	1: (* GET CLIMATIC *)
		Cmd_RLen:=20;
		FOR i:=0 TO 4 DO
			j:=DINT_TO_INT(CAL01_Clima.Points[i].X);
			TxLen:=TxLen+RAWTOHEX(ADR(j),2,ADR(TxData[TxLen]));
			j:=DINT_TO_INT(CAL01_Clima.Points[i].Y);
			TxLen:=TxLen+RAWTOHEX(ADR(j),2,ADR(TxData[TxLen]));
		END_FOR

	2: (* SET CLIMATIC *)
		IF Cmd_CLen<>20 THEN
			Cmd_R:=4;
		ELSE
			FOR i:=0 TO 4 DO
				Cmd_Buf_INT:=ADR(Cmd_Buf[8+4*i]); j:=Cmd_Buf_INT^;
				CAL01_Clima.Points[i].X:=INT_TO_DINT(j);
				Cmd_Buf_INT:=ADR(Cmd_Buf[10+4*i]); j:=Cmd_Buf_INT^;
				CAL01_Clima.Points[i].Y:=INT_TO_DINT(j);
			END_FOR
		END_IF




ELSE
	Cmd_R:=3;
END_CASE
END_ACTION
ACTION Cmd_CIR:
IF Cmd_ObjIdx<1 OR Cmd_ObjIdx>6 THEN
	Cmd_R:=2;
	RETURN;
END_IF

(* Process command *)
CASE Cmd_C OF

	1:	(* Force CIR On *)
		CASE Cmd_ObjIdx OF

		(*	1:	CIR01.CIR_RUN_REQ := TRUE; *)
			2:	CIR02.CIR_RUN_REQ := TRUE;
			3:	CIR03.CIR_RUN_REQ := TRUE;
			4:	CIR04.CIR_RUN_REQ := TRUE;
			5:	CIR05.CIR_RUN_REQ := TRUE;
			6:	CIR06.CIR_RUN_REQ := TRUE;

		END_CASE

	2:	(* Force CIR Off *)
		CASE Cmd_ObjIdx OF

		(*	1:	CIR01.CIR_STOP_REQ := TRUE; *)
			2:	CIR02.CIR_STOP_REQ := TRUE;
			3:	CIR03.CIR_STOP_REQ := TRUE;
			4:	CIR04.CIR_STOP_REQ := TRUE;
			5:	CIR05.CIR_STOP_REQ := TRUE;
			6:	CIR06.CIR_STOP_REQ := TRUE;

		END_CASE

	3:	(* Release force *)
		CASE Cmd_ObjIdx OF

		(*	1:	CIR01.CIR_RUN_REQ	:= FALSE;
				CIR01.CIR_STOP_REQ 	:= FALSE; *)
			2:	CIR02.CIR_RUN_REQ	:= FALSE;
				CIR02.CIR_STOP_REQ 	:= FALSE;
			3:	CIR03.CIR_RUN_REQ	:= FALSE;
				CIR03.CIR_STOP_REQ 	:= FALSE;
			4:	CIR04.CIR_RUN_REQ	:= FALSE;
				CIR04.CIR_STOP_REQ 	:= FALSE;
			5:	CIR05.CIR_RUN_REQ	:= FALSE;
				CIR05.CIR_STOP_REQ 	:= FALSE;
			6:	CIR06.CIR_RUN_REQ	:= FALSE;
				CIR06.CIR_STOP_REQ 	:= FALSE;

		END_CASE


	4: (* SET Tempi delay On Off Circolatori  *)
		CASE Cmd_ObjIdx OF
		(*	1:	Cmd_Buf_U16:=ADR(Cmd_Buf[8]);
				CIR01.OnDelay := DWORD_TO_TIME((Cmd_Buf_U16^)*60*1000); 			(* Delay ON*)
				Cmd_Buf_U16:=ADR(Cmd_Buf[10]);
				CIR01.OffDelay := DWORD_TO_TIME((Cmd_Buf_U16^)*60*1000);			(* Delay OFF *) *)

			2:	Cmd_Buf_U16:=ADR(Cmd_Buf[8]);
				CIR02.OnDelay := DWORD_TO_TIME((Cmd_Buf_U16^)*60*1000);			(* Delay ON*)
				Cmd_Buf_U16:=ADR(Cmd_Buf[10]);
				CIR02.OffDelay := DWORD_TO_TIME((Cmd_Buf_U16^)*60*1000);			(* Delay OFF *)

			3:	Cmd_Buf_U16:=ADR(Cmd_Buf[8]);
				CIR03.OnDelay := DWORD_TO_TIME((Cmd_Buf_U16^)*60*1000); 			(* Delay ON*)
				Cmd_Buf_U16:=ADR(Cmd_Buf[10]);
				CIR03.OffDelay := DWORD_TO_TIME((Cmd_Buf_U16^)*60*1000);			(* Delay OFF *)

			4:	Cmd_Buf_U16:=ADR(Cmd_Buf[8]);
				CIR04.OnDelay := DWORD_TO_TIME((Cmd_Buf_U16^)*60*1000);			(* Delay ON*)
				Cmd_Buf_U16:=ADR(Cmd_Buf[10]);
				CIR04.OffDelay := DWORD_TO_TIME((Cmd_Buf_U16^)*60*1000);			(* Delay OFF *)

			5:	Cmd_Buf_U16:=ADR(Cmd_Buf[8]);
				CIR05.OnDelay := DWORD_TO_TIME((Cmd_Buf_U16^)*60*1000); 			(* Delay ON*)
				Cmd_Buf_U16:=ADR(Cmd_Buf[10]);
				CIR05.OffDelay := DWORD_TO_TIME((Cmd_Buf_U16^)*60*1000);			(* Delay OFF *)

			6:	Cmd_Buf_U16:=ADR(Cmd_Buf[8]);
				CIR06.OnDelay := DWORD_TO_TIME((Cmd_Buf_U16^)*60*1000);			(* Delay ON*)
				Cmd_Buf_U16:=ADR(Cmd_Buf[10]);
				CIR06.OffDelay := DWORD_TO_TIME((Cmd_Buf_U16^)*60*1000);			(* Delay OFF *)

		END_CASE


	5: (* GET Tempi delay On Off Circolatori *)
		Cmd_RLen:=4;
			CASE Cmd_ObjIdx OF


		(*	1:	j:=DWORD_TO_WORD(TIME_TO_DWORD((CIR01.OnDelay)/60/1000));
				TxLen:=TxLen+RAWTOHEX(ADR(j),2,ADR(TxData[TxLen]));
				j:=DWORD_TO_WORD(TIME_TO_DWORD((CIR01.OffDelay)/60/1000));
				TxLen:=TxLen+RAWTOHEX(ADR(j),2,ADR(TxData[TxLen]));   *)
			2: 	j:=DWORD_TO_WORD(TIME_TO_DWORD((CIR02.OnDelay)/60/1000));
				TxLen:=TxLen+RAWTOHEX(ADR(j),2,ADR(TxData[TxLen]));
				j:=DWORD_TO_WORD(TIME_TO_DWORD((CIR02.OffDelay)/60/1000));
				TxLen:=TxLen+RAWTOHEX(ADR(j),2,ADR(TxData[TxLen]));
			3:	j:=DWORD_TO_WORD(TIME_TO_DWORD((CIR03.OnDelay)/60/1000));
				TxLen:=TxLen+RAWTOHEX(ADR(j),2,ADR(TxData[TxLen]));
				j:=DWORD_TO_WORD(TIME_TO_DWORD((CIR03.OffDelay)/60/1000));
				TxLen:=TxLen+RAWTOHEX(ADR(j),2,ADR(TxData[TxLen]));
			4: 	j:=DWORD_TO_WORD(TIME_TO_DWORD((CIR04.OnDelay)/60/1000));
				TxLen:=TxLen+RAWTOHEX(ADR(j),2,ADR(TxData[TxLen]));
				j:=DWORD_TO_WORD(TIME_TO_DWORD((CIR04.OffDelay)/60/1000));
				TxLen:=TxLen+RAWTOHEX(ADR(j),2,ADR(TxData[TxLen]));
			5:	j:=DWORD_TO_WORD(TIME_TO_DWORD((CIR05.OnDelay)/60/1000));
				TxLen:=TxLen+RAWTOHEX(ADR(j),2,ADR(TxData[TxLen]));
				j:=DWORD_TO_WORD(TIME_TO_DWORD((CIR05.OffDelay)/60/1000));
				TxLen:=TxLen+RAWTOHEX(ADR(j),2,ADR(TxData[TxLen]));
			6: 	j:=DWORD_TO_WORD(TIME_TO_DWORD((CIR06.OnDelay)/60/1000));
				TxLen:=TxLen+RAWTOHEX(ADR(j),2,ADR(TxData[TxLen]));
				j:=DWORD_TO_WORD(TIME_TO_DWORD((CIR06.OffDelay)/60/1000));
				TxLen:=TxLen+RAWTOHEX(ADR(j),2,ADR(TxData[TxLen]));
		END_CASE










ELSE
	Cmd_R:=3;
END_CASE
END_ACTION
ACTION Cmd_CIRD:
IF Cmd_ObjIdx<1 OR Cmd_ObjIdx>2 THEN
	Cmd_R:=2;
	RETURN;
END_IF

(* Process command *)
CASE Cmd_C OF

	1:	(* Force CIR On *)
		CASE Cmd_ObjIdx OF

(*			1:	CIRD01.CIR_RUN_REQ := TRUE;
			2:	CIRD02.CIR_RUN_REQ := TRUE;
			3:	CIRD03.CIR_RUN_REQ := TRUE; *)

		END_CASE

	2:	(* Force CIR Off *)
		CASE Cmd_ObjIdx OF

(*			1:	CIRD01.CIR_STOP_REQ := TRUE;
			2:	CIRD02.CIR_STOP_REQ := TRUE;
			3:	CIRD03.CIR_STOP_REQ := TRUE; *)

		END_CASE

	3:	(* Release force *)
		CASE Cmd_ObjIdx OF

(*			1:	CIRD01.CIR_RUN_REQ	:= FALSE;
				CIRD01.CIR_STOP_REQ := FALSE;
			2:	CIRD02.CIR_RUN_REQ	:= FALSE;
				CIRD02.CIR_STOP_REQ := FALSE;
			3:	CIRD03.CIR_RUN_REQ 	:= FALSE;
				CIRD03.CIR_STOP_REQ := FALSE; *)

		END_CASE

ELSE
	Cmd_R:=3;
END_CASE
END_ACTION
ACTION Cmd_CRON:
(* Check index *)
IF Cmd_ObjIdx<1 OR Cmd_ObjIdx>6 THEN
	Cmd_R:=2;
	RETURN;
END_IF

(* Process command *)
CASE Cmd_C OF

	1: (* GET PROFILE *)
		IF Cmd_CLen<>3 THEN
			Cmd_R:=4;
		ELSE
			(* Load profile *)
			CronEd.CN_Sel:=WORD_TO_BYTE(Cmd_ObjIdx);
			Cmd_Buf_U16:=ADR(Cmd_Buf[8]);
			CronEd.CN_YSel:=Cmd_Buf_U16^;
			IF Cmd_Buf[10]<=10 THEN
				CronEd.PR_Sel:=Cmd_Buf[10];
				CronEd.PR_Load_Exe();
				(* Response data *)
				Cmd_RLen:=192;
				TxLen:=TxLen+RAWTOHEX(ADR(CronEd.PR.Setpoint),192,ADR(TxData[TxLen]));
			ELSE
				Cmd_R:=6;
			END_IF
		END_IF

	2: (* SET PROFILE *)
		IF Cmd_CLen<>(3+192) THEN
			Cmd_R:=4;
		ELSE
			(* Save profile *)
			CronEd.CN_Sel:=WORD_TO_BYTE(Cmd_ObjIdx);
			Cmd_Buf_U16:=ADR(Cmd_Buf[8]);
			CronEd.CN_YSel:=Cmd_Buf_U16^;
			IF Cmd_Buf[10]<=10 THEN
				CronEd.PR_Sel:=Cmd_Buf[10];
				MEMCPY(ADR(Cmd_Buf[11]),ADR(CronEd.PR.Setpoint),192);
				CronEd.PR_Save_Exe_Multi(); (* updated by DB - for saving profiles in eventually existing multiple crono files *)
			ELSE
				Cmd_R:=6;
			END_IF
		END_IF

	5: (* GET CALENDAR MONTH *)
		IF Cmd_CLen<>3 THEN
			Cmd_R:=4;
		ELSE
			(* Load calendar *)
			CronEd.CN_Sel:=WORD_TO_BYTE(Cmd_ObjIdx);
			Cmd_Buf_U16:=ADR(Cmd_Buf[8]);
			CronEd.CN_YSel:=Cmd_Buf_U16^;
			IF Cmd_Buf[10]>=1 AND Cmd_Buf[10]<=12 THEN
				CronEd.CA_Sel:=Cmd_Buf[10];
				CronEd.CA_Load_Exe();
				(* Response data *)
				Cmd_RLen:=32;
				TxLen:=TxLen+RAWTOHEX(ADR(CronEd.CA.Profile),32,ADR(TxData[TxLen]));
			ELSE
				Cmd_R:=6;
			END_IF
		END_IF

	6: (* SET CALENDAR MONTH *)
		IF Cmd_CLen<>(3+32) THEN
			Cmd_R:=4;
		ELSE
			(* Save calendar *)
			CronEd.CN_Sel:=WORD_TO_BYTE(Cmd_ObjIdx);
			Cmd_Buf_U16:=ADR(Cmd_Buf[8]);
			CronEd.CN_YSel:=Cmd_Buf_U16^;
			IF Cmd_Buf[10]>=1 AND Cmd_Buf[10]<=12 THEN
				CronEd.CA_Sel:=Cmd_Buf[10];
				MEMCPY(ADR(Cmd_Buf[11]),ADR(CronEd.CA.Profile),32);
				CronEd.CA_Save_Exe();
			ELSE
				Cmd_R:=6;
			END_IF
		END_IF

	9: (* CRON RESTART *)
		CASE Cmd_ObjIdx OF
			1: THER01.InitOK:=FALSE;
			2: THER02.InitOK:=FALSE;
			3: THER03.InitOK:=FALSE;
			4: THER04.InitOK:=FALSE;
			5: THER05.InitOK:=FALSE;
			6: THER06.InitOK:=FALSE;
		END_CASE

	10: (* SET Isteresi  *)
		CASE Cmd_ObjIdx OF
			1:	Cmd_Buf_U16:=ADR(Cmd_Buf[8]);
				THER01.Histeresys := Cmd_Buf_U16^; 			(* Isteresi*)
			2:	Cmd_Buf_U16:=ADR(Cmd_Buf[8]);
				THER02.Histeresys := Cmd_Buf_U16^; 			(* Isteresi*)
			3:	Cmd_Buf_U16:=ADR(Cmd_Buf[8]);
				THER03.Histeresys := Cmd_Buf_U16^; 			(* Isteresi*)
			4:	Cmd_Buf_U16:=ADR(Cmd_Buf[8]);
				THER04.Histeresys := Cmd_Buf_U16^; 			(* Isteresi*)
			5:	Cmd_Buf_U16:=ADR(Cmd_Buf[8]);
				THER05.Histeresys := Cmd_Buf_U16^; 			(* Isteresi*)
			6:	Cmd_Buf_U16:=ADR(Cmd_Buf[8]);
				THER06.Histeresys := Cmd_Buf_U16^; 			(* Isteresi*)

		END_CASE

	11: (* GET isteresi *)
		Cmd_RLen:=2;
		CASE Cmd_ObjIdx OF


			1: j:=(THER01.Histeresys);
				TxLen:=TxLen+RAWTOHEX(ADR(j),2,ADR(TxData[TxLen]));
			2: j:=(THER02.Histeresys);
				TxLen:=TxLen+RAWTOHEX(ADR(j),2,ADR(TxData[TxLen]));
			3: j:=(THER03.Histeresys);
				TxLen:=TxLen+RAWTOHEX(ADR(j),2,ADR(TxData[TxLen]));
			4: j:=(THER04.Histeresys);
				TxLen:=TxLen+RAWTOHEX(ADR(j),2,ADR(TxData[TxLen]));
			5: j:=(THER05.Histeresys);
				TxLen:=TxLen+RAWTOHEX(ADR(j),2,ADR(TxData[TxLen]));
			6: j:=(THER06.Histeresys);
				TxLen:=TxLen+RAWTOHEX(ADR(j),2,ADR(TxData[TxLen]));

		END_CASE











ELSE
	Cmd_R:=3;
END_CASE
END_ACTION
ACTION Cmd_GRU:
(* Check index *)(*
IF Cmd_ObjIdx<>1 THEN
	Cmd_R:=2;
	RETURN;
END_IF

(* Process command *)
CASE Cmd_C OF

	1: (* GET CLIMATIC *)
		Cmd_RLen:=20;
		FOR i:=0 TO 4 DO
			j:=DINT_TO_INT(GRU01_Clima.Points[i].X);
			TxLen:=TxLen+RAWTOHEX(ADR(j),2,ADR(TxData[TxLen]));
			j:=DINT_TO_INT(GRU01_Clima.Points[i].Y);
			TxLen:=TxLen+RAWTOHEX(ADR(j),2,ADR(TxData[TxLen]));
		END_FOR

	2: (* SET CLIMATIC *)
		IF Cmd_CLen<>20 THEN
			Cmd_R:=4;
		ELSE
			FOR i:=0 TO 4 DO
				Cmd_Buf_INT:=ADR(Cmd_Buf[8+4*i]); j:=Cmd_Buf_INT^;
				GRU01_Clima.Points[i].X:=INT_TO_DINT(j);
				Cmd_Buf_INT:=ADR(Cmd_Buf[10+4*i]); j:=Cmd_Buf_INT^;
				GRU01_Clima.Points[i].Y:=INT_TO_DINT(j);
			END_FOR
		END_IF

ELSE
	Cmd_R:=3;
END_CASE
*);
END_ACTION
ACTION Cmd_PDC:
(* Check index *)
IF Cmd_ObjIdx<>1 THEN
	Cmd_R:=2;
	RETURN;
END_IF

(* Process command *)
CASE Cmd_C OF

	1: (* GET CLIMATIC *)
		Cmd_RLen:=20;
		FOR i:=0 TO 4 DO
			j:=DINT_TO_INT(PDC01_Clima.Points[i].X);
			TxLen:=TxLen+RAWTOHEX(ADR(j),2,ADR(TxData[TxLen]));
			j:=DINT_TO_INT(PDC01_Clima.Points[i].Y);
			TxLen:=TxLen+RAWTOHEX(ADR(j),2,ADR(TxData[TxLen]));
		END_FOR

	2: (* SET CLIMATIC *)
		IF Cmd_CLen<>20 THEN
			Cmd_R:=4;
		ELSE
			FOR i:=0 TO 4 DO
				Cmd_Buf_INT:=ADR(Cmd_Buf[8+4*i]); j:=Cmd_Buf_INT^;
				PDC01_Clima.Points[i].X:=(j);(*INT_TO_DINT(j); *)
				Cmd_Buf_INT:=ADR(Cmd_Buf[10+4*i]); j:=Cmd_Buf_INT^;
				PDC01_Clima.Points[i].Y:=(j); (*INT_TO_DINT(j); *)
			END_FOR
		END_IF


	3:	(* Force On *)
		CASE Cmd_ObjIdx OF

			1:	PDC01.RUN_REQ := TRUE;
				PDC01.STOP_REQ := FALSE;

		END_CASE

	4:	(* Force Off *)
		CASE Cmd_ObjIdx OF

			1:	PDC01.STOP_REQ := TRUE;
				PDC01.RUN_REQ := FALSE;

		END_CASE

	5:	(* Release force *)
		CASE Cmd_ObjIdx OF

			1:	PDC01.RUN_REQ	:= FALSE;
				PDC01.STOP_REQ := FALSE;

		END_CASE

	6: (* SET Tempi delay On Off   *)
		CASE Cmd_ObjIdx OF
			1:	Cmd_Buf_U16:=ADR(Cmd_Buf[8]);
				PDC01.OnDelay := DWORD_TO_TIME((Cmd_Buf_U16^)*60*1000); 			(* Delay ON*)
				Cmd_Buf_U16:=ADR(Cmd_Buf[10]);
				PDC01.OffDelay := DWORD_TO_TIME((Cmd_Buf_U16^)*60*1000);			(* Delay OFF *)

		END_CASE


	7: (* GET Tempi delay On Off  *)
		Cmd_RLen:=4;
			CASE Cmd_ObjIdx OF


			1:	j:=DWORD_TO_WORD(TIME_TO_DWORD((PDC01.OnDelay)/60/1000));
				TxLen:=TxLen+RAWTOHEX(ADR(j),2,ADR(TxData[TxLen]));
				j:=DWORD_TO_WORD(TIME_TO_DWORD((PDC01.OffDelay)/60/1000));
				TxLen:=TxLen+RAWTOHEX(ADR(j),2,ADR(TxData[TxLen]));

			END_CASE

(*	8: (* SET Comandi  *)
		CASE Cmd_ObjIdx OF
			1:	Cmd_Buf_U16:=ADR(Cmd_Buf[8]);
				PDC01.PDCbilitata := DWORD_TO_BOOL(Cmd_Buf_U16^); 	(* Chiller Abilitato 0=Disabilitato   1=abilitato *)
				Cmd_Buf_U16:=ADR(Cmd_Buf[10]);
				PDC01.ImpMB_ResetFrigo := DWORD_TO_BOOL(Cmd_Buf_U16^); (* Comando reset sicurezze1=RESET  *)
				Cmd_Buf_U16:=ADR(Cmd_Buf[12]);
				PDC01.ImpMB_LocRem := DWORD_TO_BOOL(Cmd_Buf_U16^); 	(* Comando locale/remoto (toggle)0=LOCALE   1=REMOTO  *)

				PDC01.fWriteAttivazioneComandi:= TRUE;		(* da abilitare mettendo a true - abilitazione scrittura variabile Modbus *)
				PDC01.Refresh_Now := TRUE;

		END_CASE



	9: (* GET Comandi  *)
		Cmd_RLen:=6;
			CASE Cmd_ObjIdx OF


			1:	j:=BOOL_TO_INT(PDC01.PDCbilitata);
				TxLen:=TxLen+RAWTOHEX(ADR(j),2,ADR(TxData[TxLen]));
				j:=BOOL_TO_INT(PDC01.MB_BitStato[2]);				(* Comando reset sicurezze1=RESET  *)
				TxLen:=TxLen+RAWTOHEX(ADR(j),2,ADR(TxData[TxLen]));
				j:=BOOL_TO_INT(PDC01.MB_BitStato[3]);				(* Comando locale/remoto (toggle)0=LOCALE   1=REMOTO  *)
				TxLen:=TxLen+RAWTOHEX(ADR(j),2,ADR(TxData[TxLen]));

       	END_CASE
*)


	10: (* SET Comandi  *)
		CASE Cmd_ObjIdx OF
			1:	Cmd_Buf_U16:=ADR(Cmd_Buf[8]);
				PDC01.ScriviCoil := DWORD_TO_BOOL(Cmd_Buf_U16^); 	(* 0 write on register - 1 write on coil *)
				Cmd_Buf_U16:=ADR(Cmd_Buf[10]);
				PDC01.IndirizzoDaScrivere :=(Cmd_Buf_U16^); 		(* Address of the register / coil.  *)
				Cmd_Buf_U16:=ADR(Cmd_Buf[12]);
				PDC01.DatoDaScrivere := (Cmd_Buf_U16^); 			(* The value to be written.  *)

				PDC01.ScriviDato:= TRUE;							(* da abilitare mettendo a true - abilitazione scrittura variabile Modbus *)
				PDC01.Refresh_Now := TRUE;

		END_CASE






ELSE
	Cmd_R:=3;
END_CASE
END_ACTION
ACTION Cmd_SYS:
(* Check index *)
IF Cmd_ObjIdx<>0 THEN
	Cmd_R:=2;
	RETURN;
END_IF

(* Process command *)
CASE Cmd_C OF

	0: (* ECHO *)
		IF Cmd_CLen<>0 THEN
			TxLen:=0;
		END_IF

	1: (* LOG REQUEST *)
		LogTrig();

	2: (* REARM *)
		Sys.Warning:=FALSE;
		Sys.Alarm:=FALSE;
		Sys.AlarmStop:=FALSE;

	3: (* GET INFO1 *)
		Cmd_RLen:=6;
		TxLen:=TxLen+RAWTOHEX(ADR(Plant_SN),4,ADR(TxData[TxLen]));
		TxLen:=TxLen+RAWTOHEX(ADR(Plant_SW_VER),2,ADR(TxData[TxLen]));

	4: (*  Scrivo i Parametri gestione Impianto   *)

			Cmd_Buf_U16:=ADR(Cmd_Buf[8]);
			DelayAllarmeTemperaturaNonRaggiunta := Cmd_Buf_U16^; 			(* Ritardo Allarme dall'avvio Caldaia*)
			Cmd_Buf_U16:=ADR(Cmd_Buf[10]);
			DeltaInterventoAllarmeTempeaturaNonRaggiuta := Cmd_Buf_U16^;	(* Delta Soglia Temperatura per Allarme Temperatura Non Raggiunta *)
			Cmd_Buf_U16:=ADR(Cmd_Buf[12]);
			OffsetSetPointManuale := Cmd_Buf_U16^; 							(* Offest Perdite Scambiatore 1  *)
			Cmd_Buf_U16:=ADR(Cmd_Buf[14]);
			OffsetSetPointManuale2 := Cmd_Buf_U16^; 						(* Offest Perdite Scambiatore 1  *)
			Cmd_Buf_U16:=ADR(Cmd_Buf[12]);
			BitAbilitaBoost :=INT_TO_BOOL( Cmd_Buf_U16^); 					(* Abilitazione controllo Boost  *)
			Cmd_Buf_U16:=ADR(Cmd_Buf[14]);
			RifOffsetBoost := Cmd_Buf_U16^; 								(* Offset al Setpoint della Caldaia per azione di Boost  *)


	5: (*  Leggi i parametri gestione Impianto  *)

			Cmd_RLen:=18;
			j:=(DelayAllarmeTemperaturaNonRaggiunta);   				(* Ritardo Allarme dall'avvio Caldaia*)
			TxLen:=TxLen+RAWTOHEX(ADR(j),2,ADR(TxData[TxLen]));
			j:=(DeltaInterventoAllarmeTempeaturaNonRaggiuta);			(* Delta Soglia Temperatura per Allarme Temperatura Non Raggiunta *)
			TxLen:=TxLen+RAWTOHEX(ADR(j),2,ADR(TxData[TxLen]));
			j:=(OffsetSetPointManuale);									(* Offest Perdite Scambiatore 1  *)
			TxLen:=TxLen+RAWTOHEX(ADR(j),2,ADR(TxData[TxLen]));
			j:=(OffsetSetPointManuale2);								(* Offest Perdite Scambiatore 2  *)
			TxLen:=TxLen+RAWTOHEX(ADR(j),2,ADR(TxData[TxLen]));
			j:=BOOL_TO_INT(BitAbilitaBoost);							(* Abilitazione controllo Boost  *)
			TxLen:=TxLen+RAWTOHEX(ADR(j),2,ADR(TxData[TxLen]));
			j:=BOOL_TO_INT(BitAbilitaBoost);										(* Offset al Setpoint della Caldaia per azione di Boost   *)
			TxLen:=TxLen+RAWTOHEX(ADR(j),2,ADR(TxData[TxLen]));




	6: (*  Scrivo i Parametri gestione Impianto - Antigelo   *)

			Cmd_Buf_U16:=ADR(Cmd_Buf[8]);
			SogliaMinStartAntigelo := Cmd_Buf_U16^; 			(* Soglia mininma Start Antigelo *)
			Cmd_Buf_U16:=ADR(Cmd_Buf[10]);
			SogliaMinStopAntigelo := Cmd_Buf_U16^;				(* Soglia Massima Stop Antigelo *)
			Cmd_Buf_U16:=ADR(Cmd_Buf[12]);
			BitAbilitaAntigelo :=INT_TO_BOOL( Cmd_Buf_U16^); 	(* Abilitazione Antigelo  *)

	7: (*  Leggi i parametri gestione Impianto - Antigelo *)

			Cmd_RLen:=14;
			j:=(SogliaMinStartAntigelo); 							(* Soglia mininma Start Antigelo *)
			TxLen:=TxLen+RAWTOHEX(ADR(j),2,ADR(TxData[TxLen]));
			j:=(SogliaMinStopAntigelo);								(* Soglia Massima Stop Antigelo *)
			TxLen:=TxLen+RAWTOHEX(ADR(j),2,ADR(TxData[TxLen]));
			j:=BOOL_TO_INT(BitAbilitaAntigelo);						(* Abilitazione Antigelo  *)
			TxLen:=TxLen+RAWTOHEX(ADR(j),2,ADR(TxData[TxLen]));

(*	10: (*  Scrivo i Parametri per la gestione della velocità dei circolatori sui primari   *)

			Cmd_Buf_U16:=ADR(Cmd_Buf[8]);
			PercVelMin := Cmd_Buf_U16^;
			Cmd_Buf_U16:=ADR(Cmd_Buf[10]);
			PercVelMax := Cmd_Buf_U16^;
			Cmd_Buf_U16:=ADR(Cmd_Buf[12]);
			ErroreTempMax := Cmd_Buf_U16^;
			Cmd_Buf_U16:=ADR(Cmd_Buf[14]);
			ErroreTempMin := Cmd_Buf_U16^;

	11: (*  Leggo i Parametri per la gestione della velocità dei circolatori sui primari   *)

			Cmd_RLen:=8;
			j:=(PercVelMin);
			TxLen:=TxLen+RAWTOHEX(ADR(j),2,ADR(TxData[TxLen]));
			j:=(PercVelMax);
			TxLen:=TxLen+RAWTOHEX(ADR(j),2,ADR(TxData[TxLen]));
			j:=(ErroreTempMax);
			TxLen:=TxLen+RAWTOHEX(ADR(j),2,ADR(TxData[TxLen]));
			j:=(ErroreTempMin);
			TxLen:=TxLen+RAWTOHEX(ADR(j),2,ADR(TxData[TxLen]));


	12: (*  Scrivo i Parametri per la gestione della velocità dei circolatori sui primari   *)


				Cmd_Buf_U16:=ADR(Cmd_Buf[8]);
				CAS01.DeltaTempThr := Cmd_Buf_U16^;
				Cmd_Buf_U16:=ADR(Cmd_Buf[10]);
				CAS01.Tmonitor_Off := DWORD_TO_TIME((Cmd_Buf_U16^)*60*1000);
				Cmd_Buf_U16:=ADR(Cmd_Buf[12]);
				CAS01.Tmonitor_On := DWORD_TO_TIME((Cmd_Buf_U16^)*60*1000);

	13: (*  Leggo i Parametri per la gestione della velocità dei circolatori sui primari   *)


				Cmd_RLen:=6;
				j:=(CAS01.DeltaTempThr);
				TxLen:=TxLen+RAWTOHEX(ADR(j),2,ADR(TxData[TxLen]));
				j:=DWORD_TO_WORD(TIME_TO_DWORD((CAS01.Tmonitor_Off)/60/1000));
				TxLen:=TxLen+RAWTOHEX(ADR(j),2,ADR(TxData[TxLen]));
				j:=DWORD_TO_WORD(TIME_TO_DWORD((CAS01.Tmonitor_On)/60/1000));
				TxLen:=TxLen+RAWTOHEX(ADR(j),2,ADR(TxData[TxLen]));


*)


	14: (*  Imposto data e ora del PLC  *)


			Cmd_Buf_U16:=ADR(Cmd_Buf[8]);
			SetAnno:= Cmd_Buf_U16^; 												(* Anno *)
			Cmd_Buf_U16:=ADR(Cmd_Buf[10]);
			SetMese:= Cmd_Buf_U16^;												 	(* mese *)
			Cmd_Buf_U16:=ADR(Cmd_Buf[12]);
			SetGiorno:=( Cmd_Buf_U16^);											 	(* Giorno *)
			Cmd_Buf_U16:=ADR(Cmd_Buf[14]);
			SetOra:=( Cmd_Buf_U16^); 												(* ora *)
			Cmd_Buf_U16:=ADR(Cmd_Buf[16]);
			SetMinuti:= ( Cmd_Buf_U16^);										 	(* Minuti *)
			Cmd_Buf_U16:=ADR(Cmd_Buf[18]);
			SetSecondi:= ( Cmd_Buf_U16^);										 	(* secondi *)

	(*		SysRtcSetTime(SetDataTime(DWORD_TO_INT(ADR(Cmd_Buf[8])),				(* Anno *)
										DWORD_TO_INT(ADR(Cmd_Buf[10])),				(* mese *)
										DWORD_TO_INT(ADR(Cmd_Buf[11])),				(* Giorno *)
										DWORD_TO_INT(ADR(Cmd_Buf[12])),				(* ora *)
										DWORD_TO_INT(ADR(Cmd_Buf[13])),				(* Minuti *)
										DWORD_TO_INT(ADR(Cmd_Buf[14]))				(* secondi *)
										)); *)

		SysRtcSetTime((SetDataTime(SetAnno,SetMese,SetGiorno,SetOra,SetMinuti,SetSecondi)));




ELSE
	Cmd_R:=3;
END_CASE
END_ACTION
ACTION Cmd_VRD:
(* Check index *)
IF Cmd_ObjIdx<1 OR Cmd_ObjIdx>2 THEN
	Cmd_R:=2;
	RETURN;
END_IF

(* Process command *)
CASE Cmd_C OF

	1: (* GET CLIMATIC *)
		Cmd_RLen:=20;
		FOR i:=0 TO 4 DO
			IF Cmd_ObjIdx=1 THEN
				j:=DINT_TO_INT(VRD01_Clima.Points[i].X);
			ELSE
				j:=DINT_TO_INT(VRD02_Clima.Points[i].X);
			END_IF
			TxLen:=TxLen+RAWTOHEX(ADR(j),2,ADR(TxData[TxLen]));
			IF Cmd_ObjIdx=1 THEN
				j:=DINT_TO_INT(VRD01_Clima.Points[i].Y);
			ELSE
				j:=DINT_TO_INT(VRD02_Clima.Points[i].Y);
			END_IF
			TxLen:=TxLen+RAWTOHEX(ADR(j),2,ADR(TxData[TxLen]));
		END_FOR

	2: (* SET CLIMATIC *)
		IF Cmd_CLen<>20 THEN
			Cmd_R:=4;
		ELSE
			FOR i:=0 TO 4 DO
				Cmd_Buf_INT:=ADR(Cmd_Buf[8+4*i]); j:=Cmd_Buf_INT^;
				IF Cmd_ObjIdx=1 THEN
					VRD01_Clima.Points[i].X:=INT_TO_DINT(j);
				ELSE
					VRD02_Clima.Points[i].X:=INT_TO_DINT(j);
				END_IF
				Cmd_Buf_INT:=ADR(Cmd_Buf[10+4*i]); j:=Cmd_Buf_INT^;
				IF Cmd_ObjIdx=1 THEN
					VRD01_Clima.Points[i].Y:=INT_TO_DINT(j);
				ELSE
					VRD02_Clima.Points[i].Y:=INT_TO_DINT(j);
				END_IF
			END_FOR
		END_IF

ELSE
	Cmd_R:=3;
END_CASE
END_ACTION
ACTION Command:
(* Default response OK/NODATA *)
Cmd_R:=0;
Cmd_RLen:=0;
TxLen:=16;

(* Check object *)
CASE Cmd_Obj OF

	EO_SYS:
		Cmd_SYS();
(*
	EO_GRU:
		Cmd_GRU();

	EO_PDC:
		Cmd_PDC();
*)
	EO_CAL:
		Cmd_CAL();

	EO_CRON, EO_THER:
		Cmd_CRON();

	EO_VRD:
		Cmd_VRD();

	EO_CIR:
		Cmd_CIR();

(*	EO_CIRD,EO_CIRDM:
		Cmd_CIRD();
*)

ELSE
	Cmd_R:=1;
END_CASE

(* Generate response *)
IF TxLen>0 THEN
	RAWTOHEX(ADR(Cmd_Obj)	,2,ADR(TxData[ 0]));
	RAWTOHEX(ADR(Cmd_ObjIdx),2,ADR(TxData[ 4]));
	RAWTOHEX(ADR(Cmd_R)		,2,ADR(TxData[ 8]));
	RAWTOHEX(ADR(Cmd_RLen)	,2,ADR(TxData[12]));
	TxTrig:=TRUE;
END_IF
END_ACTION

(* POU Utils Functions/TCPSERVER, ST *)
FUNCTION_BLOCK TCPSERVER
(***********************************************************************************************************	*)
(* Version: 1.6                                    			          											*)
(* Date: 11.02.2011                                   					          							    *)
(***********************************************************************************************************	*)
(* WAGO Kontakttechnik GmbH Hansastr. 27 32423 Minden(Westf.)													*)
(* Tel. +0049 571/887-0 Fax. +0049 571/887-0																	*)
(* Author: VB																									*)
(***********************************************************************************************************	*)
(*Description:	A TCP server to read and write data													       		*)
(*Historie:																										*)
(*Version 1.6: 11.02.2011: Changes according to 750-880/881											 			*)
(*Version 1.5: 27.11.2008 Bugfix allow reuse port																*)
(*Version 1.4: 13.10.2008 Bugfix transmitting large data														*)
(*Version 1.3: 15.01.2007 Changes according to FW11																*)
(*Version 1.2: 09.03.2006 Changes for socket handle 0											       			*)
(*Version 1.1: 14.02.2005 Release																				*)
(***********************************************************************************************************	*)
VAR CONSTANT
	STATE_INIT     				 : BYTE:= 0;
	STATE_OPEN     				 : BYTE:= 1;
	STATE_TX       				 : BYTE:= 20;
	STATE_RX       				 : BYTE:= 30;
	STATE_CLOSE    				 : BYTE:= 40;
	STATE_ERROR_TRAP		 	 : BYTE:= 200;
END_VAR
VAR_INPUT
	xEnable    					: BOOL;	 (* Set TRUE to enable function block *)
	wPortNumber					: WORD;  (* Port *)
	tServerTimeOut				: TIME:=t#50s;
	ptSendData					: POINTER TO ARRAY[0..MAX_SEND_TCP_SERVER] OF BYTE;
	diSendCount					: DINT;
END_VAR
VAR_OUTPUT
	xClientConnected  			: BOOL:= FALSE;
	diError 					: DINT:= 0;
END_VAR
(* Status Codes -----------------------------------------
	16#8001 => No socket descriptor available 
	16#8002 => SysSockBind fails 
	16#8003 => SysSockListen fails 
	16#8004 => switching to none blocking mode fails
	16#8005 => SysSockClose() returns FALSE 
    16#8006 => SysSockConnect() fails
    16#8007 => SysSockSend() fails
	16#8008 => error state machine 
	16#8009 => timeout while waiting for data from server 
	16#0001 => server waiting for client to establish connection
------------------------------------------------------------*)
VAR_IN_OUT
	xStartSend					: BOOL;
	aReceiveBuffer				: ARRAY [0..MAX_RECEIVE_TCP_SERVER] OF BYTE;
	diReceiveCount				: DINT;
END_VAR

VAR
	m_State    					: BYTE:= 0;
	m_ReceiveBuffer				: ARRAY [0..MAX_RECEIVE_TCP_SERVER_SOCKET] OF BYTE;
	m_ServerSocket				: DINT:= SOCKET_INVALID;
	m_Socket					: DINT:= SOCKET_INVALID;
	m_AddressInfo				: SOCKADDRESS;
	m_BytesReceived				: DINT;
	m_diReturn					: DINT;
	m_xReturn					: BOOL;
	m_SizeSockadr				: DWORD;
	m_ConnectionWatchdog		: TON;
	m_Flags						: DINT;
	m_NoneBlocking   			: DINT:= 1;
	m_Blocking   				: DINT:= 0;
	i							: INT;
	m_count						: DINT;
	diOption					: DINT := 1;
	on: DINT;
END_VAR
IF xEnable THEN
	CASE m_State OF
		STATE_INIT:
			(* Create Socket *)
			m_ServerSocket:= SysSockCreate( SOCKET_AF_INET, SOCKET_STREAM, 0);
			IF m_ServerSocket = SOCKET_INVALID THEN
				(* *)
				diError:= 16#8001;
				m_State:= STATE_ERROR_TRAP;
				RETURN;
			ELSE
				;
			END_IF
			(* Address bindings *)
			(********************)
			on:=1;
			SysSockSetOption( m_ServerSocket, SOCKET_SOL, SOCKET_SO_REUSEADDR, ADR(on), SIZEOF(on) );

			m_AddressInfo.sin_family:= SOCKET_AF_INET;
			m_AddressInfo.sin_port  := SysSockHtons( wPortNumber);
			m_AddressInfo.sin_addr  := SOCKET_INADDR_ANY;
			IF NOT SysSockBind( m_ServerSocket, ADR(m_AddressInfo), SIZEOF(m_AddressInfo)) THEN
				diError:= 16#8002;
				m_State:= STATE_ERROR_TRAP;
				RETURN;
			END_IF
			(* Wait for connections *)
			(************************)
			IF NOT SysSockListen( m_ServerSocket, 1) THEN
				diError:= 16#8003;
				m_State:= STATE_ERROR_TRAP;
			END_IF

			(* Puts SOCKET in NonBlocking mode *)
			m_diReturn:= SysSockIoctl( m_ServerSocket, SOCKET_FIONBIO, ADR(m_NoneBlocking));

			m_State:= STATE_OPEN;


		STATE_OPEN: 	(* Waiting for incomming connection *)
				m_SizeSockadr:=SIZEOF(m_AddressInfo);
				m_Socket:= SysSockAccept( m_ServerSocket, ADR(m_AddressInfo), ADR(m_SizeSockadr));
				diError:=State_open;
				IF m_Socket <> SOCKET_INVALID THEN
					xClientConnected:=TRUE;
					(*Set Push-Bit:new V1.5*)
					IF ADR(%MW0)=16#30000000  OR ADR(%MW0)=16#20000000 THEN (*841 or 881*)
						SysSockSetOption(
							diSocket:=m_Socket,
							diLevel:=6,
							diOption:=SOCKET_TCP_NODELAY,
							pOptionValue:=ADR(diOption),
							diOptionLength:=SIZEOF(diOption));
					ELSE
							;
					END_IF
					SysSockIoctl( m_Socket, SOCKET_FIONBIO, ADR(m_NoneBlocking));
					m_State:= STATE_RX;
					diError:=0;
				END_IF

		STATE_RX:
					m_BytesReceived:= SysSockRecv( m_Socket, ADR(m_ReceiveBuffer), SIZEOF(m_ReceiveBuffer), 0);
					CASE m_BytesReceived OF
					-1:(*no data available or error occured*)
						m_ConnectionWatchdog(IN:=TRUE , PT:=tServerTimeOut );
						IF m_connectionWatchdog.Q THEN
							m_State:= STATE_CLOSE;
							m_ConnectionWatchdog(IN:=FALSE);(*reset connection watchdog*)
							diError := 16#8009;
						END_IF
					0:(* socket was "gracefully closed"  *)
						m_State:= STATE_CLOSE;
						diError := 16#8003;
					ELSE
						(* Copy received data into receive buffer *)
						(********************************)
						FOR i:= 0 TO DINT_TO_INT(m_BytesReceived	)-1 DO
							aReceiveBuffer[diReceiveCount]:= m_ReceiveBuffer[i];
							diReceiveCount:=(diReceiveCount+1) MOD SIZEOF(aReceiveBuffer);
						END_FOR

						m_ConnectionWatchdog(IN:=FALSE);(*reset connection watchdog*)
					END_CASE

				(*send data*)
				IF xStartSend	 THEN
					m_State := STATE_TX;
				END_IF

	STATE_TX:	 (* send TCP-message *)
		m_diReturn := SysSockSend(diSocket := m_Socket,
								  pbyBuffer := ADR(ptSendData^[m_count]),(*geändert V1.4 bisher: [0] *)
								  diBufferSize := diSendCount-m_count,
								  diFlags :=m_Flags);
		CASE m_diReturn OF
		-1:	(* ERROR or data could not yet be send (V1.3 due to new FW11) *)
			m_ConnectionWatchdog(IN:=TRUE , PT:=tServerTimeOut );
			IF m_connectionWatchdog.Q THEN
				m_State:= STATE_CLOSE;
				m_ConnectionWatchdog(IN:=FALSE);(*reset connection watchdog*)
				diError := 16#8007;
			END_IF
		0: (* socket was "gracefully closed"  *)
			m_State := STATE_CLOSE;
			diError := 16#8003;
		ELSE (* succesful *)
			m_count:=m_count+m_diReturn;
			IF m_count>=diSendCount THEN
				diError := 16#0000;
				m_State := STATE_RX;
				m_count:=0;
				xStartSend:=FALSE;
			END_IF
			m_ConnectionWatchdog(IN:=FALSE);(*reset connection watchdog*)
		END_CASE


		STATE_CLOSE:	(* Close the server *)

		IF ADR(%MW0)=16#30000000  OR ADR(%MW0)=16#20000000 THEN (*841 or 881*)
			;
		ELSE
			IF m_Socket>=0 THEN
				SysSockShutdown(m_Socket, 0);;(*870*)
			END_IF
		END_IF
		IF m_Socket>=0 THEN
			SysSockClose( m_Socket);
		END_IF
		xClientConnected:= FALSE;
		m_State:= STATE_OPEN; (* Try to open the server again *)
		m_ConnectionWatchdog(IN:=FALSE);(*reset connection watchdog*)

		STATE_ERROR_TRAP: (* Error Read/Write socket  *)
			m_State:= STATE_ERROR_TRAP;

	ELSE  (* Bad FSM code trap  *)
			m_State:= STATE_ERROR_TRAP;
			diError:= 16#8008;
	END_CASE;
ELSE
	IF m_State <> STATE_INIT THEN
		IF ADR(%MW0)=16#30000000  OR ADR(%MW0)=16#20000000 THEN (*841 or 881*)
			;
		ELSE
			IF m_Socket>=0 THEN
				SysSockShutdown(m_Socket, 0);;(*870*)
			END_IF
		END_IF
		IF m_Socket>=0 THEN
			SysSockClose( m_Socket);
		END_IF
		IF ADR(%MW0)=16#30000000  OR ADR(%MW0)=16#20000000 THEN (*841 or 881*)
			;
		ELSE
			IF m_ServerSocket>=0 THEN
				SysSockShutdown(m_ServerSocket, 0);;(*870*)
			END_IF
		END_IF
		IF m_ServerSocket>=0 THEN
			SysSockClose( m_ServerSocket);
		END_IF
		xClientConnected:= FALSE;
		diError:= 0;
		m_State:= STATE_init; (* Try to open the server again *)
		m_ConnectionWatchdog(IN:=FALSE);(*reset connection watchdog*)
	END_IF
END_IF
END_FUNCTION_BLOCK

(* POU Utils Functions/HEXTORAW, ST *)
FUNCTION HEXTORAW : WORD
VAR_INPUT
	pString		: POINTER TO BYTE;
	StringLen	: WORD;
	pData		: POINTER TO BYTE;
END_VAR
VAR
	xl: WORD;
	xi: WORD;
	xr: BYTE;
END_VAR
xl:=0;
xi:=0;

WHILE xi<StringLen DO

	IF pString^>=97 AND pString^<=102 THEN
		xr := pString^ - 87;
	ELSIF pString^>=65 AND pString^<=70 THEN
		xr := pString^ - 55;
	ELSIF pString^>=48 AND pString^<=57 THEN
		xr := pString^ - 48;
	ELSE
		xr := 16;
	END_IF

	IF xr<16 THEN
		IF (xi AND 1)=0 THEN
			pData^ := xr * 16;
		ELSE
			pData^ := pData^ + xr;
			pData := pData + 1;
			xl := xl + 1;
		END_IF
	END_IF

	xi := xi + 1;
	pString := pString + 1;

END_WHILE

HEXTORAW:=xl;
END_FUNCTION

(* POU Utils Functions/RAWTOHEX, ST *)
FUNCTION RAWTOHEX : WORD
VAR_INPUT
	pData: POINTER TO BYTE;
	DataLen: WORD;
	pString: POINTER TO BYTE;
END_VAR
VAR
	xl: WORD;
END_VAR
xl:=0;

WHILE DataLen>0 DO

	pString^ := (pData^ / 16#10) + 48 + (((pData^ / 16#10)/10)*7);
	pString:=pString+1;
	pString^ := (pData^ AND 16#0F)  + 48 + (((pData^ AND 16#0F)/10)*7);
	pString:=pString+1;
	pData:=pData+1;
	DataLen:=DataLen-1;
	xl:=xl+2;

END_WHILE

(*pString^:=0;*)

RAWTOHEX:=xl;
END_FUNCTION

(* POU Utils Functions/GestioneDataTime_DaOscat/SetDataTime, ST *)
FUNCTION SetDataTime : DT
VAR_INPUT
	year : INT;
	month : INT;
	day : INT;
	hour : INT;
	minute : INT;
	second : INT;
END_VAR

VAR
	count : INT;
END_VAR
(* Creazione variabiletipo DT per creare Orario da dare al PLC *)


IF month > 2 THEN
	count := (month - 1) * 30;
	IF month > 7 THEN count := count + SHR(month - 3,1); ELSE count := count + SHR(month - 4,1); END_IF;
	(* chech for leap year and add one day if true *)
	IF SHL(year,14) = 0 THEN count := count + 1; END_IF;
ELSE
	count := (month - 1) * 31;
END_IF;


SetDataTime := DWORD_TO_DT(DATE_TO_DWORD( DWORD_TO_DATE((INT_TO_DWORD(count + day - 1) + SHR(INT_TO_DWORD(year) * 1461 - 2878169, 2)) * 86400))
				+ INT_TO_DWORD(SECOND)
				+ INT_TO_DWORD(MINUTE) * 60
				+ INT_TO_DWORD(HOUR) * 3600);
END_FUNCTION

(* POU Utils/CSV_Log, ST *)
FUNCTION CSV_Log : BOOL
VAR_INPUT
END_VAR
VAR CONSTANT
	LogFileName:STRING:='S:\LOGS_ID4V3.CSV';
END_VAR
VAR
	s1 : STRING(256);
	hFile: 	DWORD;
END_VAR
(* Check file presence *)
hFile:=SysFileOpen(LogFileName,'r');
IF hFile=0 THEN
	(*** File not exist *** Create file and write header *)
	hFile:=SysFileOpen(LogFileName,'w');
	IF hFile<>0 THEN
		(* Write CSV header *)
		s1:='Title1;Title2,...';
		SysFileWrite(hFile, ADR(s1), LEN(s1));
		SysFileWrite(hFile, ADR(Logger_CRLF), LEN(Logger_CRLF));
	END_IF
ELSE
	(*** File exist *** Close file and reopen in append mode *)
	SysFileClose(hFile);
	hFile:=SysFileOpen(LogFileName,'a');
END_IF

(* Log to file *)
IF hFile<>0 THEN
	(* Date stamp *)
	s1:=REPLACE( Sys.Time_LogString , ' ' , 1 , 11 );
	SysFileWrite(hFile, ADR(s1), LEN(s1));
	(* Write CSV data *)
	s1:=CONCAT(';', 'Data1' );
	s1:=CONCAT(s1 , ';');
	s1:=CONCAT(s1 , 'Data2' );
	s1:=CONCAT(s1 , ';');
	s1:=CONCAT(s1 , '...' );
	SysFileWrite(hFile, ADR(s1), LEN(s1));
	(* Add line CRLF and close *)
	SysFileWrite(hFile, ADR(Logger_CRLF), LEN(Logger_CRLF));
	SysFileClose(hFile);
END_IF
END_FUNCTION

(* POU Plant/SYS_Proc, ST *)
PROGRAM SYS_Proc
VAR
(*	fALARM_PB		:FLT_TAP;
	fALARM_TB		:FLT_TAP;
	fALARM_PM		:FLT_TAP;	*)
	fALARM_ALARM_PM_PB_TB		:FLT_TAP;


(*	fGZB_ST			:FLT_TAP;  (* GATEWAY ZIGBEE *)*)
	fVPN_ST1		:FLT_TAP;  (* VPN CONNECT *)
(*	fVPN_ST2		:FLT_TAP;  (* VPN STATUS *)*)
(*	fKEY_CT_ST		:FLT_TAP;  (* DOOR1 *)*)
(*	fKEY_SCT_ST		:FLT_TAP;  (* DOOR2 *)*)
	fKEY_QE_ST		:FLT_TAP;  (* DOOR3 *)


	fBostAttivo	:FLT_TAP;

	fALARM_MancatoRaggiungimentoAcqua		:FLT_TAP;
	DelayfALARM_MancatoRaggiungimentoAcqua:TON;



END_VAR
(*************** ISPESL *****************)

fALARM_ALARM_PM_PB_TB(IN:=NOT ALARM_PM_PB_TB);
IF fALARM_ALARM_PM_PB_TB.EVH THEN
	LogEv(EL_AlarmStop,EO_PMV,1,1,'Allarmi_ISPESL');
END_IF

(*
fALARM_TB(IN:=ALARM_TB);
IF fALARM_TB.EVH THEN
	LogEv(EL_AlarmStop,EO_TBV,1,1,'Over_Temperature_Alarm');
END_IF

fALARM_PM(IN:=ALARM_PM);
IF fALARM_PM.EVH THEN
	LogEv(EL_AlarmStop,EO_PMV,1,1,'Under_Pressure_Alarm');
END_IF
*)
(****************************************)

(*### VPN Connection Check ###*)
fVPN_ST1(IN:=VPN_ST1);
IF fVPN_ST1.EVH THEN
	LogEv(EL_Log,EO_VPN,1,1,'CONNECT_ON');
END_IF
IF fVPN_ST1.EVL THEN
	LogEv(EL_Log,EO_VPN,1,2,'CONNECT_OFF');
END_IF

(*
(*### VPN Status Check ###*)
fVPN_ST2(IN:=VPN_ST2);
IF fVPN_ST2.EVH THEN
	LogEv(EL_Log,EO_VPN,1,3,'STATUS_UP');
END_IF
IF fVPN_ST2.EVL THEN
	LogEv(EL_Wrn,EO_VPN,1,4,'STATUS_DOWN');
END_IF
*)
(*### DOOR01 Status Check ###*)(*
fKEY_CT_ST(IN:=KEY_CT_ST);
IF fKEY_CT_ST.EVH THEN
	LogEv(EL_Log,EO_DOOR,1,2,'Centrale_termica_Close');
END_IF
IF fKEY_CT_ST.EVL THEN
	LogEv(EL_Wrn,EO_DOOR,1,1,'Centrale_termica_Open');
END_IF*)

(*### DOOR02 Status Check ###*)(*
fKEY_SCT_ST(IN:=KEY_SCT_ST);
IF fKEY_SCT_ST.EVH THEN
	LogEv(EL_Log,EO_DOOR,2,2,'Sottocentrale_termica_Close');
END_IF
IF fKEY_SCT_ST.EVL THEN
	LogEv(EL_Wrn,EO_DOOR,2,1,'Sottocentrale_termica_Open');
END_IF*)

(*### DOOR03 Status Check ###*)
fKEY_QE_ST(IN:=KEY_QE_ST);
IF fKEY_QE_ST.EVH THEN
	LogEv(EL_Log,EO_DOOR,3,2,'Quadro_Close');
END_IF
IF fKEY_QE_ST.EVL THEN
	LogEv(EL_Wrn,EO_DOOR,3,1,'Quadro_Open');
END_IF




(* ##### Allarme mancata Raggiungimento temperatura su mandata Acqua ####### *)


DelayfALARM_MancatoRaggiungimentoAcqua(IN:=(CAL01.Run),PT:=DINT_TO_TIME(DelayAllarmeTemperaturaNonRaggiunta*60000));

 (* in questo caso il delta viene applicato al Set point fisico che si da alla caldaia *)

fALARM_MancatoRaggiungimentoAcqua(IN:=DelayfALARM_MancatoRaggiungimentoAcqua.Q
									AND ( TPV02.AVG < (CAL01.nvoTempBoiler.wSnvtTemp-2740) -  DeltaInterventoAllarmeTempeaturaNonRaggiuta));
IF fALARM_MancatoRaggiungimentoAcqua.EVH THEN
	LogEv(EL_AlarmStop,EO_SYS,0,11,'Mancato_Raggiungimento_Temp');
END_IF

(* Segnalazione Boost Attivo *)

fBostAttivo(IN:=BitAbilitaBoost AND (THER250.SetPoint>TPV08.AVG));
IF fBostAttivo.EVH THEN
	LogEv(EL_Log,EO_SYS,0,14,'Boost_Attivo');
END_IF
IF fBostAttivo.EVL THEN
	LogEv(EL_Log,EO_SYS,0,15,'Boost_Non_Attivo');
END_IF
END_PROGRAM

(* POU TCP_Logger/LogEv, ST *)
FUNCTION LogEv : BOOL
VAR_INPUT
	Level	: en_Logger_ErrLev;
	Object  : en_SYS_Objects;
	Index	: WORD;
	Error	: WORD;
	Message : STRING;
END_VAR
VAR
	s1 : STRING(160);
	i  : INT;
END_VAR
(* Execute error level operations *)
CASE Level OF
	EL_Wrn: 		Sys.Warning:=TRUE;
	EL_Alarm: 		Sys.Alarm  :=TRUE;
	EL_AlarmStop: 	Sys.Alarm  :=TRUE; (* GO TO STOP STATE!! *)
END_CASE

(* Fill lastlog list *)
s1:=CONCAT(Sys.Time_LogString,';Lev=');
s1:=CONCAT(s1,INT_TO_STRING(Level));
s1:=CONCAT(s1,';Obj=');
s1:=CONCAT(s1,INT_TO_STRING(Object));
s1:=CONCAT(s1,';Idx=');
s1:=CONCAT(s1,WORD_TO_STRING(Index));
s1:=CONCAT(s1,';Err=');
s1:=CONCAT(s1,WORD_TO_STRING(Error));
Sys.LastLogs_Dat[Sys.LastLogs_Idx]:=s1;
Sys.LastLogs_Msg[Sys.LastLogs_Idx]:=Message;
Sys.LastLogs_Idx:=Sys.LastLogs_Idx+1;
IF Sys.LastLogs_Idx>5 THEN Sys.LastLogs_Idx:=0; END_IF

(*---------------------------------------------------------------*)
	Logger_Head();
(*---------------------------------------------------------------*)

(* Insert ERR *)
s1:=CONCAT('&ERR=',INT_TO_STRING(Level));
s1:=CONCAT(s1,';');
s1:=CONCAT(s1,INT_TO_STRING(Object));
s1:=CONCAT(s1,';');
s1:=CONCAT(s1,WORD_TO_STRING(Index));
s1:=CONCAT(s1,';');
s1:=CONCAT(s1,WORD_TO_STRING(Error));
s1:=CONCAT(s1,';');
ADDSTRING(ADR(Logger.TData), ADR(s1), Logger.TLen);
s1:=Message;
STR_NOSPACES(ADR(s1));
ADDSTRING(ADR(Logger.TData), ADR(s1), Logger.TLen);

(*---------------------------------------------------------------*)
	Logger_Send();
(*---------------------------------------------------------------*)
END_FUNCTION

(* POU TCP_Logger/Logger_Head, ST *)
FUNCTION Logger_Head : BOOL
VAR
	s1 : STRING(160);
	i  : BYTE;
END_VAR
Logger.TLen:=0;
(* Set GET header *)
ADDSTRING(ADR(Logger.TData), ADR(Logger_GETSTART), Logger.TLen);

(* Insert Header *)
s1:=INSERT('ID=&V=1&D=',DWORD_TO_STRING(Plant_SN),3);
s1:=CONCAT(s1,REPLACE(Sys.Time_LogString,'T',1,11));
s1:=CONCAT(s1,'&S=');
IF Sys.Alarm THEN i:=2; ELSIF Sys.Warning THEN i:=1; ELSE i:=0; END_IF
s1:=CONCAT(s1,BYTE_TO_STRING(i));
ADDSTRING(ADR(Logger.TData), ADR(s1), Logger.TLen);
END_FUNCTION

(* POU Utils Functions/ADDSTRING, ST *)
FUNCTION ADDSTRING : BOOL (* Append string to a byte buffer *)
VAR_INPUT
	pTxData: POINTER TO BYTE;
	pString: POINTER TO BYTE;
END_VAR
VAR_IN_OUT
	TxLen: DINT;
END_VAR
VAR
END_VAR
pTxData:=pTxData+TxLen;
WHILE pString^<>0 DO
	pTxData^:=pString^;
	pString:=pString+1;
	pTxData:=pTxData+1;
	TxLen:=TxLen+1;
END_WHILE
END_FUNCTION

(* POU Utils Functions/STR_NOSPACES, ST *)
FUNCTION STR_NOSPACES : BOOL (* Replace spaces and bad chars with allowed ones, used as HTTP-GET validator *)
VAR_INPUT
	pString: POINTER TO BYTE;
END_VAR
VAR
END_VAR
WHILE pString^<>0 DO
	IF pString^=16#20 (* space *) THEN pString^:=16#5F; (*'_'*) END_IF
	pString:=pString+1;
END_WHILE
END_FUNCTION

(* POU TCP_Logger/Logger_Send, ST *)
FUNCTION Logger_Send : BOOL
VAR
	hFile: 	DWORD;
	pos:	DWORD;
END_VAR
(* Finalize string *)
ADDSTRING(ADR(Logger.TData), ADR(Logger_GETEND), Logger.TLen);

(* Read log position *)
pos:=SysFileGetSize(Logger_DataFile);
(* Check log size, bckup and erase if no pending messages *)
IF pos>5000000(*5M*) THEN
	hFile:=SysFileOpen(Logger_IndexFile,'r');
	IF hFile=0 THEN
		SysFileDelete(Logger_DataFileOld);
		SysFileRename(Logger_DataFile,Logger_DataFileOld);
		pos:=0;
	ELSE
		SysFileClose(hFile);
	END_IF
END_IF
(* Write message on log file *)
hFile:=SysFileOpen(Logger_DataFile,'a');
IF hFile<>0 THEN
	SysFileWrite(hFile, ADR(Logger.TData), Logger.TLen);
	SysFileClose(hFile);
ELSE
	Sys.Warning:=TRUE;
END_IF


(* Check logger status *)
IF Logger.SendReq=FALSE THEN
	(* Set log position for recovery *)
	Logger.SendIdx:=pos;
	(* Copy message data *)
	MEMCPY(ADR(Logger.TData),ADR(Logger.SendData),DINT_TO_WORD(Logger.TLen));
	Logger.SendLen:=Logger.TLen;
	(* Trigger request *)
	Logger.SendReq:=TRUE;
ELSE
	(* Add message position+size in recovery indexes *)
	hFile:=SysFileOpen(Logger_IndexFile,'a');
	SysFileWrite(hFile, ADR(pos), SIZEOF(pos));
	SysFileWrite(hFile, ADR(Logger.TLen), SIZEOF(Logger.TLen));
	SysFileClose(hFile);
END_IF
END_FUNCTION

(* POU Utils Functions/MEMCPY, ST *)
FUNCTION MEMCPY:BOOL
VAR_INPUT
	pSourceAddress:POINTER TO ARRAY[1..2] OF BYTE;
	pDestinationAddress:POINTER TO ARRAY[1..2] OF BYTE;
	BytesToCopy:WORD;
END_VAR
VAR
END_VAR
WHILE (BytesToCopy > 0) DO
	pDestinationAddress^[1]:=pSourceAddress^[1]; (* copy bytes from source to destination *)
	pDestinationAddress:=ADR(pDestinationAddress^[2]); (* increment destination *)
	pSourceAddress:=ADR(pSourceAddress^[2]);(* increment source *)
	BytesToCopy:=BytesToCopy -1; (* decrement number of bytes to copy *)
END_WHILE
END_FUNCTION

(* POU Utils Functions/AVERAGE_DINT, ST *)
FUNCTION_BLOCK AVERAGE_DINT
VAR_INPUT
	IN: 	DINT;
END_VAR
VAR_OUTPUT
	HI:		DINT;
	AVG:	DINT;
	LOW:	DINT;
	ERR:	BOOL;
END_VAR
VAR
	sum:	REAL;
	cnt:	WORD;
END_VAR
IF cnt>=65000 THEN
	ERR:=TRUE;
	Read();
	sum := sum - DINT_TO_REAL(AVG);
	cnt := cnt - 1;
END_IF

sum := sum + DINT_TO_REAL(IN);
cnt := cnt + 1;

IF IN<LOW THEN LOW:=IN; END_IF
IF IN>HI  THEN HI :=IN; END_IF
END_FUNCTION_BLOCK
ACTION Read:
AVG := REAL_TO_DINT(sum/cnt);
END_ACTION
ACTION Reset:
HI:=IN;
AVG:=IN;
LOW:=IN;
ERR:=FALSE;

sum:=DINT_TO_REAL(IN);
cnt:=1;
END_ACTION

(* POU Utils Functions/AVERAGE_INT, ST *)
FUNCTION_BLOCK AVERAGE_INT
VAR_INPUT
	IN: 	INT;
END_VAR
VAR_OUTPUT
	HI:		INT;
	AVG:	INT;
	LOW:	INT;
	ERR:	BOOL;
END_VAR
VAR
	sum:	DINT;
	cnt:	WORD;
END_VAR
IF cnt>=65000 THEN
	ERR:=TRUE;
	Read();
	sum := sum - AVG;
	cnt := cnt - 1;
END_IF

sum := sum + IN;
cnt := cnt + 1;

IF IN<LOW THEN LOW:=IN; END_IF
IF IN>HI  THEN HI :=IN; END_IF
END_FUNCTION_BLOCK
ACTION Read:
AVG := DINT_TO_INT(sum/cnt);
END_ACTION
ACTION Reset:
HI:=IN;
AVG:=IN;
LOW:=IN;
ERR:=FALSE;

sum:=IN;
cnt:=1;
END_ACTION

(* POU Utils Functions/AVERAGE_T, ST *)
FUNCTION_BLOCK AVERAGE_T
VAR_INPUT
	IN: 	INT;
END_VAR
VAR_OUTPUT
	HI:		INT;
	AVG:	INT;
	LOW:	INT;
	ERR:	BOOL;
END_VAR
VAR
	sum:	DINT;
	cnt:	WORD;
END_VAR
IF cnt>=65000 THEN
	ERR:=TRUE;
	Read();
	sum := sum - AVG;
	cnt := cnt + 1;
END_IF

sum := sum + IN;
cnt := cnt + 1;

IF IN<LOW THEN  LOW:=IN; END_IF
IF IN>HI  THEN HI :=IN; END_IF
END_FUNCTION_BLOCK
ACTION Read:
AVG := DINT_TO_INT(sum/cnt);
END_ACTION
ACTION Reset:
HI:=IN;
AVG:=IN;
LOW:=IN;
ERR:=FALSE;

sum:=IN;
cnt:=1;
END_ACTION

(* POU Utils Functions/BUILD_16TO32, ST *)
FUNCTION BUILD_16TO32 : DWORD
VAR_INPUT
		pSource	:	POINTER TO WORD;
END_VAR
VAR
		Data	:	DWORD;
END_VAR
Data := WORD_TO_DWORD(pSource^);
pSource := pSource + 1;
Data := Data + WORD_TO_DWORD(pSource^) * 65536;

BUILD_16TO32 := Data;
END_FUNCTION

(* POU Utils Functions/COPY_32SWAP16, ST *)
FUNCTION COPY_32SWAP16:BOOL
VAR_INPUT
	pSourceAddress		:POINTER TO ARRAY[1..2] OF WORD;
	pDestinationAddress	:POINTER TO ARRAY[1..2] OF WORD;
END_VAR
VAR
END_VAR
pDestinationAddress^[1]:=pSourceAddress^[2];
pDestinationAddress^[2]:=pSourceAddress^[1];
END_FUNCTION

(* POU LON/Shared/Type scaling functions/FbDecodeSnvtLevPercent, ST *)
FUNCTION_BLOCK FbDecodeSnvtLevPercent
VAR_INPUT
	value : typSnvtLevPercent;
END_VAR
VAR_OUTPUT
	rScaledValue : REAL;
END_VAR
VAR
END_VAR
rScaledValue := INT_TO_REAL(value.iSnvtLevPercent) / 200;
END_FUNCTION_BLOCK

(* POU LON/Shared/Type scaling functions/FbDecodeSnvtSwitch, ST *)
FUNCTION_BLOCK FbDecodeSnvtSwitch
VAR_INPUT
	value : typSnvtSwitch;
END_VAR
VAR_OUTPUT
	rValue : REAL;
	xState : BOOL;
END_VAR
VAR
END_VAR
rValue := BYTE_TO_REAL(value.bValue) / 2;
xState := (value.siState > 0);
END_FUNCTION_BLOCK

(* POU LON/Shared/Type scaling functions/FbDecodeSnvtTemp, ST *)
FUNCTION_BLOCK FbDecodeSnvtTemp
VAR_INPUT
	value : typSnvtTemp;
END_VAR
VAR_OUTPUT
	rScaledValue : REAL;
END_VAR
VAR
END_VAR
rScaledValue := (WORD_TO_REAL(value.wSnvtTemp) - 2740.0) / 10.0;
END_FUNCTION_BLOCK

(* POU LON/Shared/Type scaling functions/FbDecodeSnvtTempP, ST *)
FUNCTION_BLOCK FbDecodeSnvtTempP
VAR_INPUT
	value : typSnvtTempP;
END_VAR
VAR_OUTPUT
	rScaledValue : REAL;
END_VAR
VAR
END_VAR
rScaledValue := INT_TO_REAL(value.iSnvtTempP) / 100;
END_FUNCTION_BLOCK

(* POU Utils Functions/FLT_EVENT, ST *)
FUNCTION_BLOCK FLT_EVENT
VAR_INPUT
	IN		: BOOL;
	INITEV	: BOOL:=TRUE;
END_VAR
VAR_OUTPUT
	EVH		: BOOL;
	EVL		: BOOL;
END_VAR
VAR
	init	: BOOL:=FALSE;
	old		: BOOL;
END_VAR
EVH:=FALSE;
EVL:=FALSE;

IF NOT init THEN
	init:=TRUE;
	IF INITEV THEN
		old := NOT IN;
	ELSE
		old := IN;
	END_IF
END_IF

IF old<>IN THEN
	old:=IN;
	IF IN THEN EVH:=TRUE; ELSE EVL:=TRUE; END_IF
END_IF
END_FUNCTION_BLOCK

(* POU Utils Functions/FLT_TIME, ST *)
FUNCTION_BLOCK FLT_TIME
VAR_INPUT
	IN		: BOOL;
	TTAP	: TIME:=T#5s;
	INITEV	: BOOL:=TRUE;
END_VAR
VAR_OUTPUT
	OUT		: BOOL;
	EVH		: BOOL;
	EVL		: BOOL;
END_VAR
VAR
	init	: BOOL:=FALSE;
	timer	: TON;
END_VAR
EVH:=FALSE;
EVL:=FALSE;

IF NOT init THEN
	init := TRUE;
	IF INITEV THEN
		OUT  := NOT IN;
	ELSE
		OUT  := IN;
	END_IF
END_IF

IF OUT<>IN THEN
	timer(IN:=TRUE,PT:=TTAP);
	IF timer.Q THEN
		OUT:=IN;
		timer(IN:=FALSE);
		IF OUT THEN EVH:=TRUE; ELSE EVL:=TRUE; END_IF
	END_IF
ELSE
	timer(IN:=FALSE);
END_IF
END_FUNCTION_BLOCK

(* POU LON/Module_1/Internal/FuDoCpUpdate_Module_1, ST *)
FUNCTION FuDoCpUpdate_Module_1 : BOOL
(******************************************)
(* Automatic generated code, do not edit! *)
(******************************************)
VAR_INPUT
	ptCp : POINTER TO BYTE;
	ptCpLast : POINTER TO BYTE;
	wCpIndex : WORD;
	uiCpLength : UINT;
	uiCpVariableLength : UINT;
END_VAR
OutDataTelegram_Module_1[0] := C2M_CP_VALUE;
OutDataTelegram_Module_1[1] := WORD_TO_BYTE(wCpIndex AND 16#FF);
OutDataTelegram_Module_1[2] := WORD_TO_BYTE((wCpIndex / 256) AND 16#FF);

mbxModule_1.bTxPrio := 1;
mbxModule_1.bTxProtID := 0;
mbxModule_1.pbTxData := ADR(OutDataTelegram_Module_1);
mbxModule_1.unTxLen := 3 + uiCpLength;
mbxModule_1.MBX_SEND();

IF (mbxModule_1.nError <> MBX_OK) THEN
	FuDoCpUpdate_Module_1 := FALSE;
	RETURN;
END_IF

FuMemCopy(ptCp, ptCpLast, uiCpVariableLength);

FuDoCpUpdate_Module_1 := TRUE;
END_FUNCTION

(* POU LON/Shared/Type scaling functions/FuEncodeSnvtLevPercent, ST *)
FUNCTION FuEncodeSnvtLevPercent : typSnvtLevPercent
VAR_INPUT
	rValue : REAL;
END_VAR
VAR
END_VAR
IF rValue < -163.84 THEN rValue := -163.84; END_IF
IF rValue > 163.83 THEN rValue := 163.83; END_IF
FuEncodeSnvtLevPercent.iSnvtLevPercent := REAL_TO_INT(rValue * 200);
END_FUNCTION

(* POU LON/Shared/Type scaling functions/FuEncodeSnvtSwitch, ST *)
FUNCTION FuEncodeSnvtSwitch : typSnvtSwitch
VAR_INPUT
	rValue : REAL;
	xState : BOOL;
END_VAR
VAR
END_VAR
IF rValue < 0 THEN rValue := 0; END_IF
IF rValue > 100 THEN rValue := 100; END_IF
FuEncodeSnvtSwitch.bValue := REAL_TO_BYTE(rValue * 2);
IF xState THEN
	FuEncodeSnvtSwitch.siState := 1;
ELSE
	FuEncodeSnvtSwitch.siState := 0;
END_IF
END_FUNCTION

(* POU LON/Shared/Type scaling functions/FuEncodeSnvtTemp, ST *)
FUNCTION FuEncodeSnvtTemp : typSnvtTemp
VAR_INPUT
	rValue : REAL;
END_VAR
VAR
END_VAR
IF rValue < -274.0 THEN rValue := -274.0; END_IF
IF rValue > 6279.5 THEN rValue := 6279.5; END_IF
FuEncodeSnvtTemp.wSnvtTemp := REAL_TO_WORD((rValue * 10) + 2740);
END_FUNCTION

(* POU LON/Shared/Type scaling functions/FuEncodeSnvtTempP, ST *)
FUNCTION FuEncodeSnvtTempP : typSnvtTempP
VAR_INPUT
	rValue : REAL;
END_VAR
VAR
END_VAR
IF rValue < -273.17 THEN rValue := -273.17; END_IF
IF rValue > 327.66 THEN rValue := 327.66; END_IF
FuEncodeSnvtTempP.iSnvtTempP := REAL_TO_INT(rValue * 100);
END_FUNCTION

(* POU LON/Shared/Internal/FuRawToSnvtAlarm, ST *)
FUNCTION FuRawToSnvtAlarm : BOOL
(******************************************)
(* Automatic generated code, do not edit! *)
(******************************************)
VAR_INPUT
	RawDataIn : POINTER TO ARRAY[0..28] OF BYTE;
	DataOut : POINTER TO typSnvtAlarm;
END_VAR
VAR
END_VAR
DataOut^.abLocation[0] := RawDataIn^[0];
DataOut^.abLocation[1] := RawDataIn^[1];
DataOut^.abLocation[2] := RawDataIn^[2];
DataOut^.abLocation[3] := RawDataIn^[3];
DataOut^.abLocation[4] := RawDataIn^[4];
DataOut^.abLocation[5] := RawDataIn^[5];

DataOut^.wObjectId := RawDataIn^[6] * 256 + RawDataIn^[7];

DataOut^.bAlarmType := RawDataIn^[8];

DataOut^.bPriorityLevel := RawDataIn^[9];

DataOut^.wIndexToSnvt := RawDataIn^[10] * 256 + RawDataIn^[11];

DataOut^.abValue[0] := RawDataIn^[12];
DataOut^.abValue[1] := RawDataIn^[13];
DataOut^.abValue[2] := RawDataIn^[14];
DataOut^.abValue[3] := RawDataIn^[15];

DataOut^.wYear := RawDataIn^[16] * 256 + RawDataIn^[17];

DataOut^.bMonth := RawDataIn^[18];

DataOut^.bDay := RawDataIn^[19];

DataOut^.bHour := RawDataIn^[20];

DataOut^.bMinute := RawDataIn^[21];

DataOut^.bSecond := RawDataIn^[22];

DataOut^.wMillisecond := RawDataIn^[23] * 256 + RawDataIn^[24];

DataOut^.abAlarmLimit[0] := RawDataIn^[25];
DataOut^.abAlarmLimit[1] := RawDataIn^[26];
DataOut^.abAlarmLimit[2] := RawDataIn^[27];
DataOut^.abAlarmLimit[3] := RawDataIn^[28];

FuRawToSnvtAlarm := TRUE;
END_FUNCTION

(* POU LON/Shared/Internal/FuRawToSnvtCount, ST *)
FUNCTION FuRawToSnvtCount : BOOL
(******************************************)
(* Automatic generated code, do not edit! *)
(******************************************)
VAR_INPUT
	RawDataIn : POINTER TO ARRAY[0..1] OF BYTE;
	DataOut : POINTER TO typSnvtCount;
END_VAR
VAR
END_VAR
DataOut^.wSnvtCount := RawDataIn^[0] * 256 + RawDataIn^[1];

FuRawToSnvtCount := TRUE;
END_FUNCTION

(* POU LON/Shared/Internal/FuRawToSnvtFilePos, ST *)
FUNCTION FuRawToSnvtFilePos : BOOL
(******************************************)
(* Automatic generated code, do not edit! *)
(******************************************)
VAR_INPUT
	RawDataIn : POINTER TO ARRAY[0..5] OF BYTE;
	DataOut : POINTER TO typSnvtFilePos;
END_VAR
VAR
END_VAR
DataOut^.diRwPtr := RawDataIn^[0] * 16777216 + RawDataIn^[1] * 65536 + RawDataIn^[2] * 256 + RawDataIn^[3];

DataOut^.wRwLength := RawDataIn^[4] * 256 + RawDataIn^[5];

FuRawToSnvtFilePos := TRUE;
END_FUNCTION

(* POU LON/Shared/Internal/FuRawToSnvtFileReq, ST *)
FUNCTION FuRawToSnvtFileReq : BOOL
(******************************************)
(* Automatic generated code, do not edit! *)
(******************************************)
VAR_INPUT
	RawDataIn : POINTER TO ARRAY[0..11] OF BYTE;
	DataOut : POINTER TO typSnvtFileReq;
END_VAR
VAR
END_VAR
DataOut^.bRequest := RawDataIn^[0];

DataOut^.wIndex := RawDataIn^[1] * 256 + RawDataIn^[2];

DataOut^.wReceiveTimeout := RawDataIn^[3] * 256 + RawDataIn^[4];

DataOut^.abDestAddress[0] := RawDataIn^[5];
DataOut^.abDestAddress[1] := RawDataIn^[6];
DataOut^.abDestAddress[2] := RawDataIn^[7];
DataOut^.abDestAddress[3] := RawDataIn^[8];
DataOut^.abDestAddress[4] := RawDataIn^[9];

DataOut^.bAuthOn := RawDataIn^[10];

DataOut^.bPrioOn := RawDataIn^[11];

FuRawToSnvtFileReq := TRUE;
END_FUNCTION

(* POU LON/Shared/Internal/FuRawToSnvtFileStatus, ST *)
FUNCTION FuRawToSnvtFileStatus : BOOL
(******************************************)
(* Automatic generated code, do not edit! *)
(******************************************)
VAR_INPUT
	RawDataIn : POINTER TO ARRAY[0..26] OF BYTE;
	DataOut : POINTER TO typSnvtFileStatus;
END_VAR
VAR
END_VAR
DataOut^.bStatus := RawDataIn^[0];

DataOut^.wNumberOfFiles := RawDataIn^[1] * 256 + RawDataIn^[2];

DataOut^.wSelectedFile := RawDataIn^[3] * 256 + RawDataIn^[4];

DataOut^.abAdr[0] := RawDataIn^[5];
DataOut^.abAdr[1] := RawDataIn^[6];
DataOut^.abAdr[2] := RawDataIn^[7];
DataOut^.abAdr[3] := RawDataIn^[8];
DataOut^.abAdr[4] := RawDataIn^[9];
DataOut^.abAdr[5] := RawDataIn^[10];
DataOut^.abAdr[6] := RawDataIn^[11];
DataOut^.abAdr[7] := RawDataIn^[12];
DataOut^.abAdr[8] := RawDataIn^[13];
DataOut^.abAdr[9] := RawDataIn^[14];
DataOut^.abAdr[10] := RawDataIn^[15];
DataOut^.abAdr[11] := RawDataIn^[16];
DataOut^.abAdr[12] := RawDataIn^[17];
DataOut^.abAdr[13] := RawDataIn^[18];
DataOut^.abAdr[14] := RawDataIn^[19];
DataOut^.abAdr[15] := RawDataIn^[20];
DataOut^.abAdr[16] := RawDataIn^[21];
DataOut^.abAdr[17] := RawDataIn^[22];
DataOut^.abAdr[18] := RawDataIn^[23];
DataOut^.abAdr[19] := RawDataIn^[24];
DataOut^.abAdr[20] := RawDataIn^[25];
DataOut^.abAdr[21] := RawDataIn^[26];

FuRawToSnvtFileStatus := TRUE;
END_FUNCTION

(* POU LON/Shared/Internal/FuRawToSnvtHvacMode, ST *)
FUNCTION FuRawToSnvtHvacMode : BOOL
(******************************************)
(* Automatic generated code, do not edit! *)
(******************************************)
VAR_INPUT
	RawDataIn : POINTER TO ARRAY[0..0] OF BYTE;
	DataOut : POINTER TO typSnvtHvacMode;
END_VAR
VAR
END_VAR
DataOut^.bSnvtHvacMode := RawDataIn^[0];

FuRawToSnvtHvacMode := TRUE;
END_FUNCTION

(* POU LON/Shared/Internal/FuRawToSnvtLevPercent, ST *)
FUNCTION FuRawToSnvtLevPercent : BOOL
(******************************************)
(* Automatic generated code, do not edit! *)
(******************************************)
VAR_INPUT
	RawDataIn : POINTER TO ARRAY[0..1] OF BYTE;
	DataOut : POINTER TO typSnvtLevPercent;
END_VAR
VAR
END_VAR
DataOut^.iSnvtLevPercent := RawDataIn^[0] * 256 + RawDataIn^[1];

FuRawToSnvtLevPercent := TRUE;
END_FUNCTION

(* POU LON/Shared/Internal/FuRawToSnvtObjRequest, ST *)
FUNCTION FuRawToSnvtObjRequest : BOOL
(******************************************)
(* Automatic generated code, do not edit! *)
(******************************************)
VAR_INPUT
	RawDataIn : POINTER TO ARRAY[0..2] OF BYTE;
	DataOut : POINTER TO typSnvtObjRequest;
END_VAR
VAR
END_VAR
DataOut^.wObjectId := RawDataIn^[0] * 256 + RawDataIn^[1];

DataOut^.bObjectRequest := RawDataIn^[2];

FuRawToSnvtObjRequest := TRUE;
END_FUNCTION

(* POU LON/Shared/Internal/FuRawToSnvtObjStatus, ST *)
FUNCTION FuRawToSnvtObjStatus : BOOL
(******************************************)
(* Automatic generated code, do not edit! *)
(******************************************)
VAR_INPUT
	RawDataIn : POINTER TO ARRAY[0..5] OF BYTE;
	DataOut : POINTER TO typSnvtObjStatus;
END_VAR
VAR
END_VAR
DataOut^.wObjectId := RawDataIn^[0] * 256 + RawDataIn^[1];

DataOut^.bBitfieldByteOffset2 := RawDataIn^[2];

DataOut^.bBitfieldByteOffset3 := RawDataIn^[3];

DataOut^.bBitfieldByteOffset4 := RawDataIn^[4];

DataOut^.bBitfieldByteOffset5 := RawDataIn^[5];

FuRawToSnvtObjStatus := TRUE;
END_FUNCTION

(* POU LON/Shared/Internal/FuRawToSnvtPress, ST *)
FUNCTION FuRawToSnvtPress : BOOL
(******************************************)
(* Automatic generated code, do not edit! *)
(******************************************)
VAR_INPUT
	RawDataIn : POINTER TO ARRAY[0..1] OF BYTE;
	DataOut : POINTER TO typSnvtPress;
END_VAR
VAR
END_VAR
DataOut^.iSnvtPress := RawDataIn^[0] * 256 + RawDataIn^[1];

FuRawToSnvtPress := TRUE;
END_FUNCTION

(* POU LON/Shared/Internal/FuRawToSnvtState, ST *)
FUNCTION FuRawToSnvtState : BOOL
(******************************************)
(* Automatic generated code, do not edit! *)
(******************************************)
VAR_INPUT
	RawDataIn : POINTER TO ARRAY[0..1] OF BYTE;
	DataOut : POINTER TO typSnvtState;
END_VAR
VAR
END_VAR
DataOut^.bBitfieldByteOffset0 := RawDataIn^[0];

DataOut^.bBitfieldByteOffset1 := RawDataIn^[1];

FuRawToSnvtState := TRUE;
END_FUNCTION

(* POU LON/Shared/Internal/FuRawToSnvtSwitch, ST *)
FUNCTION FuRawToSnvtSwitch : BOOL
(******************************************)
(* Automatic generated code, do not edit! *)
(******************************************)
VAR_INPUT
	RawDataIn : POINTER TO ARRAY[0..1] OF BYTE;
	DataOut : POINTER TO typSnvtSwitch;
END_VAR
VAR
END_VAR
DataOut^.bValue := RawDataIn^[0];

DataOut^.siState := RawDataIn^[1];

FuRawToSnvtSwitch := TRUE;
END_FUNCTION

(* POU LON/Shared/Internal/FuRawToSnvtTemp, ST *)
FUNCTION FuRawToSnvtTemp : BOOL
(******************************************)
(* Automatic generated code, do not edit! *)
(******************************************)
VAR_INPUT
	RawDataIn : POINTER TO ARRAY[0..1] OF BYTE;
	DataOut : POINTER TO typSnvtTemp;
END_VAR
VAR
END_VAR
DataOut^.wSnvtTemp := RawDataIn^[0] * 256 + RawDataIn^[1];

FuRawToSnvtTemp := TRUE;
END_FUNCTION

(* POU LON/Shared/Internal/FuRawToSnvtTempP, ST *)
FUNCTION FuRawToSnvtTempP : BOOL
(******************************************)
(* Automatic generated code, do not edit! *)
(******************************************)
VAR_INPUT
	RawDataIn : POINTER TO ARRAY[0..1] OF BYTE;
	DataOut : POINTER TO typSnvtTempP;
END_VAR
VAR
END_VAR
DataOut^.iSnvtTempP := RawDataIn^[0] * 256 + RawDataIn^[1];

FuRawToSnvtTempP := TRUE;
END_FUNCTION

(* POU LON/Shared/Internal/FuRawToSnvtTimeStamp, ST *)
FUNCTION FuRawToSnvtTimeStamp : BOOL
(******************************************)
(* Automatic generated code, do not edit! *)
(******************************************)
VAR_INPUT
	RawDataIn : POINTER TO ARRAY[0..6] OF BYTE;
	DataOut : POINTER TO typSnvtTimeStamp;
END_VAR
VAR
END_VAR
DataOut^.iYear := RawDataIn^[0] * 256 + RawDataIn^[1];

DataOut^.bMonth := RawDataIn^[2];

DataOut^.bDay := RawDataIn^[3];

DataOut^.bHour := RawDataIn^[4];

DataOut^.bMinute := RawDataIn^[5];

DataOut^.bSecond := RawDataIn^[6];

FuRawToSnvtTimeStamp := TRUE;
END_FUNCTION

(* POU LON/Module_1/Internal/FuSendCpValueReq_Module_1, ST *)
FUNCTION FuSendCpValueReq_Module_1 : BOOL
(******************************************)
(* Automatic generated code, do not edit! *)
(******************************************)
VAR_INPUT
	ptCp : POINTER TO BYTE;
	ptInternalUseOnly : POINTER TO BYTE;
	wCpIndex : WORD;
END_VAR
IF (ptCp <> 0) THEN
	IF ptInternalUseOnly^.0 = TRUE THEN
		OutDataTelegram_Module_1[0] := C2M_CP_VALUE_QRY;
		OutDataTelegram_Module_1[1] := WORD_TO_BYTE(wCpIndex AND 16#FF);
		OutDataTelegram_Module_1[2] := WORD_TO_BYTE((wCpIndex / 256) AND 16#FF);

		mbxModule_1.bTxPrio := 1;
		mbxModule_1.bTxProtID := 0;
		mbxModule_1.pbTxData := ADR(OutDataTelegram_Module_1);
		mbxModule_1.unTxLen := 3;
		mbxModule_1.MBX_SEND();

		IF (mbxModule_1.nError <> MBX_OK) THEN
			FuSendCpValueReq_Module_1 := FALSE;
			RETURN;
		END_IF
		ptInternalUseOnly^.0 := FALSE;
	END_IF
END_IF

FuSendCpValueReq_Module_1 := TRUE;
END_FUNCTION

(* POU LON/Shared/Internal/FuSnvtAlarmToRaw, ST *)
FUNCTION FuSnvtAlarmToRaw : BOOL
(******************************************)
(* Automatic generated code, do not edit! *)
(******************************************)
VAR_INPUT
	NvDataIn :  POINTER TO typSnvtAlarm;
	DataOut : POINTER TO ARRAY[0..28] OF BYTE;
END_VAR
VAR
END_VAR
DataOut^[0] := NvDataIn^.abLocation[0];
DataOut^[1] := NvDataIn^.abLocation[1];
DataOut^[2] := NvDataIn^.abLocation[2];
DataOut^[3] := NvDataIn^.abLocation[3];
DataOut^[4] := NvDataIn^.abLocation[4];
DataOut^[5] := NvDataIn^.abLocation[5];

DataOut^[6] := WORD_TO_BYTE(SHR(NvDataIn^.wObjectId, 8));
DataOut^[7] := WORD_TO_BYTE(NvDataIn^.wObjectId);

DataOut^[8] := NvDataIn^.bAlarmType;

DataOut^[9] := NvDataIn^.bPriorityLevel;

DataOut^[10] := WORD_TO_BYTE(SHR(NvDataIn^.wIndexToSnvt, 8));
DataOut^[11] := WORD_TO_BYTE(NvDataIn^.wIndexToSnvt);

DataOut^[12] := NvDataIn^.abValue[0];
DataOut^[13] := NvDataIn^.abValue[1];
DataOut^[14] := NvDataIn^.abValue[2];
DataOut^[15] := NvDataIn^.abValue[3];

DataOut^[16] := WORD_TO_BYTE(SHR(NvDataIn^.wYear, 8));
DataOut^[17] := WORD_TO_BYTE(NvDataIn^.wYear);

DataOut^[18] := NvDataIn^.bMonth;

DataOut^[19] := NvDataIn^.bDay;

DataOut^[20] := NvDataIn^.bHour;

DataOut^[21] := NvDataIn^.bMinute;

DataOut^[22] := NvDataIn^.bSecond;

DataOut^[23] := WORD_TO_BYTE(SHR(NvDataIn^.wMillisecond, 8));
DataOut^[24] := WORD_TO_BYTE(NvDataIn^.wMillisecond);

DataOut^[25] := NvDataIn^.abAlarmLimit[0];
DataOut^[26] := NvDataIn^.abAlarmLimit[1];
DataOut^[27] := NvDataIn^.abAlarmLimit[2];
DataOut^[28] := NvDataIn^.abAlarmLimit[3];

FuSnvtAlarmToRaw := TRUE;
END_FUNCTION

(* POU LON/Shared/Internal/FuSnvtFilePosToRaw, ST *)
FUNCTION FuSnvtFilePosToRaw : BOOL
(******************************************)
(* Automatic generated code, do not edit! *)
(******************************************)
VAR_INPUT
	NvDataIn :  POINTER TO typSnvtFilePos;
	DataOut : POINTER TO ARRAY[0..5] OF BYTE;
END_VAR
VAR
END_VAR
DataOut^[0] := DINT_TO_BYTE(SHR(NvDataIn^.diRwPtr, 24));
DataOut^[1] := DINT_TO_BYTE(SHR(NvDataIn^.diRwPtr, 16));
DataOut^[2] := DINT_TO_BYTE(SHR(NvDataIn^.diRwPtr, 8));
DataOut^[3] := DINT_TO_BYTE(NvDataIn^.diRwPtr);

DataOut^[4] := WORD_TO_BYTE(SHR(NvDataIn^.wRwLength, 8));
DataOut^[5] := WORD_TO_BYTE(NvDataIn^.wRwLength);

FuSnvtFilePosToRaw := TRUE;
END_FUNCTION

(* POU LON/Shared/Internal/FuSnvtFileReqToRaw, ST *)
FUNCTION FuSnvtFileReqToRaw : BOOL
(******************************************)
(* Automatic generated code, do not edit! *)
(******************************************)
VAR_INPUT
	NvDataIn :  POINTER TO typSnvtFileReq;
	DataOut : POINTER TO ARRAY[0..11] OF BYTE;
END_VAR
VAR
END_VAR
DataOut^[0] := NvDataIn^.bRequest;

DataOut^[1] := WORD_TO_BYTE(SHR(NvDataIn^.wIndex, 8));
DataOut^[2] := WORD_TO_BYTE(NvDataIn^.wIndex);

DataOut^[3] := WORD_TO_BYTE(SHR(NvDataIn^.wReceiveTimeout, 8));
DataOut^[4] := WORD_TO_BYTE(NvDataIn^.wReceiveTimeout);

DataOut^[5] := NvDataIn^.abDestAddress[0];
DataOut^[6] := NvDataIn^.abDestAddress[1];
DataOut^[7] := NvDataIn^.abDestAddress[2];
DataOut^[8] := NvDataIn^.abDestAddress[3];
DataOut^[9] := NvDataIn^.abDestAddress[4];

DataOut^[10] := NvDataIn^.bAuthOn;

DataOut^[11] := NvDataIn^.bPrioOn;

FuSnvtFileReqToRaw := TRUE;
END_FUNCTION

(* POU LON/Shared/Internal/FuSnvtHvacModeToRaw, ST *)
FUNCTION FuSnvtHvacModeToRaw : BOOL
(******************************************)
(* Automatic generated code, do not edit! *)
(******************************************)
VAR_INPUT
	NvDataIn :  POINTER TO typSnvtHvacMode;
	DataOut : POINTER TO ARRAY[0..0] OF BYTE;
END_VAR
VAR
END_VAR
DataOut^[0] := NvDataIn^.bSnvtHvacMode;

FuSnvtHvacModeToRaw := TRUE;
END_FUNCTION

(* POU LON/Shared/Internal/FuSnvtLevPercentToRaw, ST *)
FUNCTION FuSnvtLevPercentToRaw : BOOL
(******************************************)
(* Automatic generated code, do not edit! *)
(******************************************)
VAR_INPUT
	NvDataIn :  POINTER TO typSnvtLevPercent;
	DataOut : POINTER TO ARRAY[0..1] OF BYTE;
END_VAR
VAR
END_VAR
DataOut^[0] := INT_TO_BYTE(SHR(NvDataIn^.iSnvtLevPercent, 8));
DataOut^[1] := INT_TO_BYTE(NvDataIn^.iSnvtLevPercent);

FuSnvtLevPercentToRaw := TRUE;
END_FUNCTION

(* POU LON/Shared/Internal/FuSnvtObjRequestToRaw, ST *)
FUNCTION FuSnvtObjRequestToRaw : BOOL
(******************************************)
(* Automatic generated code, do not edit! *)
(******************************************)
VAR_INPUT
	NvDataIn :  POINTER TO typSnvtObjRequest;
	DataOut : POINTER TO ARRAY[0..2] OF BYTE;
END_VAR
VAR
END_VAR
DataOut^[0] := WORD_TO_BYTE(SHR(NvDataIn^.wObjectId, 8));
DataOut^[1] := WORD_TO_BYTE(NvDataIn^.wObjectId);

DataOut^[2] := NvDataIn^.bObjectRequest;

FuSnvtObjRequestToRaw := TRUE;
END_FUNCTION

(* POU LON/Shared/Internal/FuSnvtPressToRaw, ST *)
FUNCTION FuSnvtPressToRaw : BOOL
(******************************************)
(* Automatic generated code, do not edit! *)
(******************************************)
VAR_INPUT
	NvDataIn :  POINTER TO typSnvtPress;
	DataOut : POINTER TO ARRAY[0..1] OF BYTE;
END_VAR
VAR
END_VAR
DataOut^[0] := INT_TO_BYTE(SHR(NvDataIn^.iSnvtPress, 8));
DataOut^[1] := INT_TO_BYTE(NvDataIn^.iSnvtPress);

FuSnvtPressToRaw := TRUE;
END_FUNCTION

(* POU LON/Shared/Internal/FuSnvtStateToRaw, ST *)
FUNCTION FuSnvtStateToRaw : BOOL
(******************************************)
(* Automatic generated code, do not edit! *)
(******************************************)
VAR_INPUT
	NvDataIn :  POINTER TO typSnvtState;
	DataOut : POINTER TO ARRAY[0..1] OF BYTE;
END_VAR
VAR
END_VAR
DataOut^[0] := NvDataIn^.bBitfieldByteOffset0;

DataOut^[1] := NvDataIn^.bBitfieldByteOffset1;

FuSnvtStateToRaw := TRUE;
END_FUNCTION

(* POU LON/Shared/Internal/FuSnvtSwitchToRaw, ST *)
FUNCTION FuSnvtSwitchToRaw : BOOL
(******************************************)
(* Automatic generated code, do not edit! *)
(******************************************)
VAR_INPUT
	NvDataIn :  POINTER TO typSnvtSwitch;
	DataOut : POINTER TO ARRAY[0..1] OF BYTE;
END_VAR
VAR
END_VAR
DataOut^[0] := NvDataIn^.bValue;

DataOut^[1] := NvDataIn^.siState;

FuSnvtSwitchToRaw := TRUE;
END_FUNCTION

(* POU LON/Shared/Internal/FuSnvtTempPToRaw, ST *)
FUNCTION FuSnvtTempPToRaw : BOOL
(******************************************)
(* Automatic generated code, do not edit! *)
(******************************************)
VAR_INPUT
	NvDataIn :  POINTER TO typSnvtTempP;
	DataOut : POINTER TO ARRAY[0..1] OF BYTE;
END_VAR
VAR
END_VAR
DataOut^[0] := INT_TO_BYTE(SHR(NvDataIn^.iSnvtTempP, 8));
DataOut^[1] := INT_TO_BYTE(NvDataIn^.iSnvtTempP);

FuSnvtTempPToRaw := TRUE;
END_FUNCTION

(* POU LON/Shared/Internal/FuSnvtTimeStampToRaw, ST *)
FUNCTION FuSnvtTimeStampToRaw : BOOL
(******************************************)
(* Automatic generated code, do not edit! *)
(******************************************)
VAR_INPUT
	NvDataIn :  POINTER TO typSnvtTimeStamp;
	DataOut : POINTER TO ARRAY[0..6] OF BYTE;
END_VAR
VAR
END_VAR
DataOut^[0] := INT_TO_BYTE(SHR(NvDataIn^.iYear, 8));
DataOut^[1] := INT_TO_BYTE(NvDataIn^.iYear);

DataOut^[2] := NvDataIn^.bMonth;

DataOut^[3] := NvDataIn^.bDay;

DataOut^[4] := NvDataIn^.bHour;

DataOut^[5] := NvDataIn^.bMinute;

DataOut^[6] := NvDataIn^.bSecond;

FuSnvtTimeStampToRaw := TRUE;
END_FUNCTION

(* POU Utils Functions/LAMP_AL_GENERALE, ST *)
FUNCTION_BLOCK LAMP_AL_GENERALE
VAR_INPUT

	Allarme: BOOL;
	Warning: BOOL;
END_VAR
VAR_OUTPUT
	SistemaOK:BOOL;
	SistemaInAllarme:BOOL;
	SistemaWarning:BOOL;
	AllarmeLampada:BOOL;
END_VAR
VAR
	Lampeggio:BLINK;
END_VAR
IF Allarme THEN       					(* Se Allarme Attivo Lucde fissa ON *)
	SistemaInAllarme:=TRUE;
	SistemaWarning:=FALSE;
	AllarmeLampada:=TRUE;
ELSIF Warning THEN					(* Se Allarme Attivo Lucde fissa pulse *)
	SistemaInAllarme:=FALSE;
	SistemaWarning:=TRUE;
	Lampeggio(ENABLE:=TRUE , TIMELOW:=t#1s , TIMEHIGH:=t#1s , OUT=>AllarmeLampada );
ELSE
	SistemaInAllarme:=FALSE;
	SistemaWarning:=FALSE;
	AllarmeLampada:=FALSE;
END_IF
END_FUNCTION_BLOCK

(* POU Utils Functions/LINEAR, ST *)
FUNCTION LINEAR : REAL (* Linear interpolation *)
VAR_INPUT
	X_In	: REAL;
	P1_X	: REAL;
	P1_Y	: REAL;
	P2_X	: REAL;
	P2_Y	: REAL;
END_VAR
VAR
END_VAR
LINEAR:=P1_Y+(((P2_Y-P1_Y)*(X_In-P1_X))/(P2_X-P1_X));
END_FUNCTION

(* POU Utils Functions/LINEAR_BAD, ST *)
FUNCTION LINEAR_BAD : INT (* Linear interpolation *)
VAR_INPUT
	PuntoMinX	: INT;
	PuntoMaxX	: INT;
	ValIn		: INT;
	PuntoMinY	: REAL;
	PuntoMaxY	: REAL;
	Decimali	: BYTE;
END_VAR
VAR
	Gain				: REAL;
	PuntoMinX_R			: REAL;
	PuntoMaxX_R			: REAL;
	Linearizzazione_R	: REAL;
END_VAR
PuntoMinX_R:=INT_TO_REAL(PuntoMinX);
PuntoMaxX_R:=INT_TO_REAL(PuntoMaxX);

Gain:=(PuntoMaxX_R-PuntoMinX_R)/(PuntoMaxY-PuntoMinY);	(* Calcolo in guadagno per la linarizzazione *)
Linearizzazione_R:=PuntoMinx+(Gain*(ValIn-PuntoMinY));	(* Ottengo il valore linearizzato *)

LINEAR_BAD:=REAL_TO_INT(Linearizzazione_R*(EXPT(10, Decimali)));  (* Ottengo intero con i decimai voluti *)
END_FUNCTION

(* POU TCP_Logger/LogTrig, ST *)
FUNCTION LogTrig : BOOL
VAR
	s1 : STRING(160);
	i  : BYTE;
END_VAR
VAR_INPUT
END_VAR
(*---------------------------------------------------------------*)
	Logger_Head();
(*---------------------------------------------------------------*)

CTL01.AddLogData(COUNT:=Ctl01_Counter);

CAL01.AddLogData(CLIM:=CAL01_Clima);

Logger.s1:='&PBV=';
Logger.s1:=CONCAT(Logger.s1,SEL(ALARM_PM_PB_TB,'0','1'));
ADDSTRING(ADR(Logger.TData), ADR(Logger.s1), Logger.TLen);

(*CIR01.AddLogData(); *)
CIR02.AddLogData();
CIR03.AddLogData();
CIR04.AddLogData();
CIR05.AddLogData();
CIR06.AddLogData();

VRD01.AddLogData(CLIM:=VRD01_Clima);
VRD02.AddLogData(CLIM:=VRD02_Clima);



TPV01.AddLogData();
TPV02.AddLogData();
TPV03.AddLogData();
TPV04.AddLogData();
TPV05.AddLogData();
TPV06.AddLogData();

TPV08.AddLogData();
TPV09.AddLogData();

TPV11.AddLogData();
TPV12.AddLogData();
TPV13.AddLogData();
TPV14.AddLogData();
TPV15.AddLogData();
TPV16.AddLogData();

THER01.AddLogData();
THER02.AddLogData();
THER03.AddLogData();
THER04.AddLogData();
THER05.AddLogData();
THER06.AddLogData();
THER250.AddLogData();

PDC01.AddLogData(CLIM:=PDC01_Clima,ModBus:=MODB01);



(*---------------------------------------------------------------*)
	Logger_Send();
(*---------------------------------------------------------------*)
END_FUNCTION

(* POU Utils Functions/MEAN_T, ST *)
FUNCTION MEAN_T : INT
VAR_INPUT
		T1		:	INT;
		T2		:	INT;

		THR_L	:	INT;
		THR_H	:	INT;
END_VAR
VAR
		Tmean	:	INT;
END_VAR
IF T1 >= THR_L AND T1 <= THR_H THEN

	IF T2 >= THR_L AND T2 <= THR_H THEN
		Tmean := (T1 + T2)/2;
	ELSE
		Tmean := T1;
	END_IF
ELSE
	IF T2 >= THR_L AND T2 <= THR_H THEN
		Tmean := T2;
	ELSE
		Tmean := 16#7FFF;	(* No valid temperature data has been passed *)
	END_IF
END_IF

MEAN_T := Tmean;
END_FUNCTION

(* POU Utils Functions/MEMCLR, ST *)
FUNCTION MEMCLR:BOOL
VAR_INPUT
	pDestinationAddress:POINTER TO ARRAY[1..2] OF BYTE;
	BytesToClear:WORD;
END_VAR
VAR
END_VAR
WHILE (BytesToClear > 0) DO
	pDestinationAddress^[1]:=0;
	pDestinationAddress:=ADR(pDestinationAddress^[2]); (* increment destination *)
	BytesToClear:=BytesToClear -1; (* decrement number of bytes to copy *)
END_WHILE
END_FUNCTION

(* POU LON/Module_1/ApplicationMessage/Module_1_ApplicationMsgSend, ST *)
FUNCTION_BLOCK Module_1_ApplicationMsgSend
(******************************************)
(* Automatic generated code, do not edit! *)
(******************************************)
VAR_INPUT
	xSend 		  : BOOL;
	abAddress     : ARRAY[0..10] OF BYTE;
	typServiceSend  : ServiceType;
	xPriority : BOOL;
	xAuthentification : BOOL;
	bMsgCodeSend  : BYTE;
	abMsgDataSend : ARRAY[0..47] OF BYTE;
	bLengthSend	  : BYTE;
END_VAR
VAR_OUTPUT
	bSendStatus   : BYTE;
END_VAR
VAR
	bAddressLength : BYTE;
	RtrigSend : R_TRIG;
END_VAR
RtrigSend(CLK:=xSend);
IF RtrigSend.Q AND (xInitRunning_Module_1 = FALSE) AND (mbxModule_1.bStatus.0) THEN
	OutDataTelegram_Module_1[0] := C2M_LON_MSG_SEND;
	OutDataTelegram_Module_1[1] := INT_TO_BYTE(typServiceSend);
	OutDataTelegram_Module_1[1].6 := xAuthentification;
	OutDataTelegram_Module_1[1].7 := xPriority;
	IF (abAddress[0] = 2) THEN
		bAddressLength := 11;
	ELSE
		bAddressLength := 5;
	END_IF
	FuMemCopy(ADR(abAddress), ADR(OutDataTelegram_Module_1[2]), bAddressLength);
	OutDataTelegram_Module_1[2+bAddressLength] := bMsgCodeSend;
	IF bLengthSend > 48 THEN bLengthSend := 48; END_IF;
	FuMemCopy(ADR(abMsgDataSend), ADR(OutDataTelegram_Module_1[2+bAddressLength+1]), bLengthSend);

	mbxModule_1.bTxPrio := BOOL_TO_BYTE(xPriority);
	mbxModule_1.bTxProtID := 0;
	mbxModule_1.pbTxData := ADR(OutDataTelegram_Module_1);
	mbxModule_1.unTxLen := 3 + bAddressLength + bLengthSend;
	mbxModule_1.MBX_SEND();

	IF (mbxModule_1.nError <> MBX_OK) THEN
		bSendStatus := 255;
	ELSE
		bSendStatus := 0;
	END_IF
END_IF
END_FUNCTION_BLOCK

(* POU LON/Module_1/ApplicationMessage/Module_1_ApplicationMsgSendRsp, ST *)
FUNCTION_BLOCK Module_1_ApplicationMsgSendRsp
(******************************************)
(* Automatic generated code, do not edit! *)
(******************************************)
VAR_INPUT
	xSend 	  : BOOL;
	bCorrelator : BYTE;
	bMsgCode  : BYTE;
	abMsgData : ARRAY[0..47] OF BYTE;
	bLength	  : BYTE;
END_VAR
VAR_OUTPUT
	bSendStatus : BYTE;
END_VAR
VAR
	RtrigSend : R_TRIG;
END_VAR
RtrigSend(CLK:=xSend);
IF RtrigSend.Q AND (xInitRunning_Module_1 = FALSE) AND (mbxModule_1.bStatus.0) THEN
	OutDataTelegram_Module_1[0] := C2M_LON_MSG_RSP_SEND;
	OutDataTelegram_Module_1[1] := bCorrelator;
	OutDataTelegram_Module_1[2] := bMsgCode;
	IF bLength > 48 THEN bLength := 48; END_IF;
	FuMemCopy(ADR(abMsgData), ADR(OutDataTelegram_Module_1[3]), bLength);

	mbxModule_1.bTxPrio := BOOL_TO_BYTE(bCorrelator.7);
	mbxModule_1.bTxProtID := 0;
	mbxModule_1.pbTxData := ADR(OutDataTelegram_Module_1);
	mbxModule_1.unTxLen := 3 + bLength;
	mbxModule_1.MBX_SEND();

	IF (mbxModule_1.nError <> MBX_OK) THEN
		bSendStatus := 255;
	ELSE
		bSendStatus := 0;
	END_IF
END_IF
END_FUNCTION_BLOCK

(* POU Plant_Objects/obj_CAL_Generica, ST *)
FUNCTION_BLOCK obj_CAL_Generica
VAR_INPUT

	(* Settings *)
	ID				: BYTE;

	(* Segnali di ingresso per interfaccia  da ingressi Digitali *)
	ALARM_CAL: BOOL;
	STATO_CAL: BOOL;
	BLOCCO_CAL: BOOL;

	AI_IN:WORD;



	(* per Gestione controolo regolazione Caldaia *)

	RUN  			: BOOL;		(* Control input *)
	TEMP 			: INT;			(* Variabile di Processo*)
	FEEDBACK	: WORD;		(* Feedback controllo  *)

	Ctrl_Init		: BOOL;
	Ctrl_SetPoint	: INT;
	Ctrl_Err		: INT;			(* Current error *)
	Ctrl_Err0		: INT; 			(* Previous error *)
	Ctrl_Accel		: REAL;		(* Derivate of error *)
	Ctrl_AccelGate  : INT:=1;		(* Derivate gate *)
	Ctrl_AccelTmr	: WORD;
	Ctrl_ErrGate	: INT:=1;		(* Error gate *)
	Ctrl_Kp			: REAL:=1;		(* Proportional factor *)
	Ctrl_Kd			: REAL:=100;  	(* Derivative factor *)
	Ctrl_Out		: REAL;

	Chk_Err			: INT;
	Chk_ErrGate		: INT:=20; 		(* Check error gate *)
	Chk_Cnt			: INT;
	Chk_CntAlarm	: INT:=60; 		(* Check error trigger 60s *)


	Plant_CAL_TMax		: INT ;				(* [.1°C]  Massima temperatura ammessa sul Set Point *)
	Plant_CAL_TDefault	: INT;				(* [.1°C] Temperatura di default in caso di errore climatica *)

	Plant_CAL_TStart		: INT:=180 ;		(* [.1°C]  Temperatura Start Caldaia sul Set Point *)


	Rearm:BOOL;

	SetPointManuale: INT; 			(* SetPoint forazato in manuale escludendo la curva di carico *)
	AbilitaSetPointManuale : BOOL ; (* Abilita il funzionamento col set point Manaule Escludendo la curva cliamtica *)
	OffsetSetPointManuale:INT;		(* Offset al Setpoint manuale per comensare lo scambiatore *)

	(* Parametri per la regolazione del PID *)



END_VAR
VAR_OUTPUT
	(* Status *)
	Status_Log	: BYTE;
	Status_Vis 	: DWORD;

	(* riferimento di uscita *)
	AO_OUT:WORD;
	DO_STOP_CALDAIA:BOOL;
	DO_START_CALDAIA:BOOL;
	DO_RIARMO:BOOL;

END_VAR
VAR_IN_OUT
	CLIM		  : typ_Clima;
END_VAR
VAR
	fALARM_CAL: FLT_TAP;
	fSTATO_CAL: FLT_TAP;
	fSTATOPosizione_CAL: FLT_TAP;

	Alarm: BOOL;
	Warning:BOOL;
	Warning2: BOOL;

	Curve 		: CHARCURVE;
	Curve_Err 	: BYTE;
	Curve_Temp	: INT;

	TP_RIARMO: TP:=(PT:=t#5s);
	SetPointCaldaia: INT;

	RegolazionePid: PID;
	HMI_RifManuale: REAL;
	HMI_PIDManuale: BOOL;

	OUT_PID: REAL;
	HMI_ResetPID: BOOL;
	errore: INT;
	TON_CheckErrorePos:TON;

END_VAR

VAR_INPUT RETAIN
	KP_PID: REAL := 10;
	TN_PID: REAL := 0;
	TV_PID: REAL := 0;
	BandaMortaPID: INT := 20;
	Tolleranza: INT:=1600;  (* la tolleranz ain questo caso è su 32766 punti quindi il 5% *)
	TempoTolleranza:DINT:=5 ;

END_VAR
(* Recupero della curva cliamtica *)
(*
IF NOT CLIM.InitOK THEN Clima_Default(); END_IF;
(* Calculate Setpoint *)
Curve(	IN:= T_AMB,	N:= 5, P:= CLIM.Points,
		OUT=> Ctrl_SetPoint, ERR=> Curve_Err );
IF Curve_Err>0  OR Ctrl_SetPoint>Plant_CAL_TMax THEN
	Ctrl_SetPoint:=Plant_CAL_TDefault;
	IF NOT Warning THEN
		Warning:=TRUE;
		LogEv(EL_Wrn,EO_CAL,ID,2,'Climatic_Error');
	END_IF
ELSE
	Warning:=FALSE;
END_IF
*)

(* Scelta del set point della cladaia o viene preso dalla curva cliamtica o da un riferimento esterno *)
IF AbilitaSetPointManuale THEN
	SetPointCaldaia:=(SetPointManuale+OffsetSetPointManuale)*10;
ELSE
	SetPointCaldaia:=Ctrl_SetPoint*10;
END_IF


(***** regolazione caldaia in funzione del Set Point appena passato con la curva Clima *************)

(* Banda Morta *)
errore:=INT_TO_UINT((TEMP )-(SetPointCaldaia));
IF errore>BandaMortaPID OR errore<(BandaMortaPID*-1) THEN

	RegolazionePid(
				ACTUAL:=INT_TO_REAL(TEMP ),
				SET_POINT:=INT_TO_REAL(SetPointCaldaia),
				KP:=KP_PID ,
				TN:=TN_PID ,
				TV:=TV_PID ,
				Y_MANUAL:=HMI_RifManuale ,
				Y_OFFSET:=0 ,
				Y_MIN:=0 ,
				Y_MAX:= 100,
				MANUAL:=HMI_PIDManuale ,
				RESET:= HMI_ResetPID,
				Y=>OUT_PID ,
				LIMITS_ACTIVE=> ,
				OVERFLOW=> );

ELSE
		HMI_PIDManuale:=TRUE;
		HMI_RifManuale:=RegolazionePid.Y;

END_IF
(* ANtibumm *)
IF RUN AND (NOT Alarm) AND NOT HMI_PIDManuale THEN
	HMI_RifManuale:=RegolazionePid.Y;
END_IF

(* Adattamento segnale Analogico per uscita WAGO *)
AO_OUT:=REAL_TO_INT(RegolazionePid.Y)*(32766-REAL_TO_INT(RegolazionePid.Y_MAX-RegolazionePid.Y_MIN));




(********** Segnalazione Allarmi  ***************)

(*Segnalzione Allarme CALDAIA *)
(*
fALARM_CAL(IN:=ALARM_CAL);
IF fALARM_CAL.EVH THEN
	IF NOT Alarm THEN
		Alarm:=TRUE;
		LogEv(EL_Alarm,EO_CAL,ID,4,'CALDAIA_IN_BLOCCO ');    (******************************segnalazione *******************************)
	END_IF
ELSE
	LogEv(EL_Log,EO_CAL,ID,1,'CALDAIA_RIARMATA');
	Alarm:=FALSE;
END_IF
*)
(* Stato CALDAIA *)
fSTATO_CAL(IN:=STATO_CAL);
IF fSTATO_CAL.EVH THEN
	LogEv(EL_Log,EO_CAL,ID,1,'CALDAIA_RUN');
END_IF
IF fSTATO_CAL.EVL THEN
	LogEv(EL_Log,EO_CAL,1,2,'CALDAIA_STOP');
END_IF

(**** Controllo Feedback Poenza Caldaia *)


(* Calculate position error according to feedback *)

Errore := AO_OUT - AI_IN;


TON_CheckErrorePos(IN:=ABS(Errore)>Tolleranza,PT:=DINT_TO_TIME(TempoTolleranza*1000)); (*  il tempo tolleranza è espresso in secondi *)

fSTATOPosizione_CAL(IN:=TON_CheckErrorePos.Q );
IF fSTATOPosizione_CAL.EVH THEN
	LogEv(EL_Alarm,EO_CAL,ID,4,'FeedBack_non_Corretto');
	Warning2:=TRUE;
END_IF
IF fSTATOPosizione_CAL.EVL THEN
	LogEv(EL_Log,EO_CAL,ID,1,'FeedBack_Corretto');
	Warning2:=FALSE;
END_IF




(*


(* Execute control loop [T=500ms] *)
IF RUN AND (NOT Alarm) THEN
	(* Calculate error *)
	Ctrl_Err:=Ctrl_SetPoint-TEMP;
	(* Init/restart operations *)
	IF NOT Ctrl_Init THEN
		Ctrl_Accel:=0;
		Ctrl_AccelTmr:=0;
		Ctrl_Err0:=Ctrl_Err;
		Ctrl_Out:=5000;
		Ctrl_Init:=TRUE;
	END_IF
	(* Calculate acceleration *)
	IF ABS(Ctrl_Err-Ctrl_Err0)>Ctrl_AccelGate OR Ctrl_AccelTmr>20 THEN
		Ctrl_Accel:=INT_TO_REAL(Ctrl_Err-Ctrl_Err0)/WORD_TO_REAL(1+Ctrl_AccelTmr);
		Ctrl_AccelTmr:=0;
		Ctrl_Err0:=Ctrl_Err;
	ELSE
		Ctrl_AccelTmr:=Ctrl_AccelTmr+1;
	END_IF
	(* Gate error *)
	IF ABS(Ctrl_Err)>Ctrl_ErrGate THEN
		(* Control loop *)
		Ctrl_Out:=Ctrl_Out+(Ctrl_Kp*Ctrl_Err)+(Ctrl_Kd*Ctrl_Accel);
	END_IF
	(* Limiter and Output *)
	Ctrl_Out:=LIMIT(0,Ctrl_Out,32767);
	AO_OUT:=REAL_TO_WORD(Ctrl_Out);
ELSE
	Ctrl_Init:=FALSE;
	AO_OUT:=0;
END_IF
*)
(* Controllo On/Off Caldaia *)
(* Set running flag *)

IF RUN AND (NOT Alarm) THEN
	DO_START_CALDAIA:=TRUE;
 ELSE
	DO_START_CALDAIA:=FALSE;
END_IF


(** Riarmo Reset Caldaia  ***)

TP_RIARMO(IN:=Rearm );
DO_RIARMO:=TP_RIARMO.Q;
Rearm:=TP_RIARMO.Q;

(* Stato CALDAIA *)
fALARM_CAL(IN:=ALARM_CAL);
IF fALARM_CAL.EVH THEN
	LogEv(EL_AlarmStop,EO_CAL,ID,4,'Caldaia_In_Blocco');
END_IF
IF fALARM_CAL.EVL THEN
	LogEv(EL_Log,EO_CAL,ID,1,'CALDAIA_Sbloccata');
END_IF




(* Seganalzione stato Caldaia *)
  IF Alarm OR BLOCCO_CAL THEN
		Status_Log:=2; Status_Vis:=16#2020F0;
		AO_OUT:=0;
	ELSIF Warning OR Warning2 THEN Status_Log:=1; Status_Vis:=16#20F0F0;
    ELSE
		Status_Log:=0;
		Status_Vis:=16#006000;
END_IF
END_FUNCTION_BLOCK
ACTION AddLogData:
Logger.s1:=INSERT('&CAL=',BYTE_TO_STRING(ID),4);
IF ID<10 THEN Logger.s1:=INSERT(Logger.s1,'0',4); END_IF

Logger.s1:=CONCAT(Logger.s1,INT_TO_STRING(SetPointCaldaia/10));				Logger.s1:=CONCAT(Logger.s1,';');
Logger.s1:=CONCAT(Logger.s1,SEL(DO_START_CALDAIA,'0','100'));				Logger.s1:=CONCAT(Logger.s1,';');

Logger.s1:=CONCAT(Logger.s1,WORD_TO_STRING(Status_Log));
(*
Logger.s1:=CONCAT(Logger.s1,';');
Logger.s1:=CONCAT(Logger.s1,INT_TO_STRING(OffsetSetPointManuale));
Logger.s1:=CONCAT(Logger.s1,';');
Logger.s1:=CONCAT(Logger.s1,INT_TO_STRING(CFD_GetEnable.bValue/2)); (* Potenza Caldaia *)
Logger.s1:=CONCAT(Logger.s1,';');
Logger.s1:=CONCAT(Logger.s1,INT_TO_STRING(CFD_GetEnable.siState)); 	(* Presenza Fiamma *)
Logger.s1:=CONCAT(Logger.s1,';');
Logger.s1:=CONCAT(Logger.s1,INT_TO_STRING(CFD_Temp.iSnvtTempP/10)); 	(* Temp. Mandata da Caldaia*)
*)


ADDSTRING(ADR(Logger.TData), ADR(Logger.s1), Logger.TLen);
END_ACTION
ACTION Clima_Default:
CLIM.Points[0].X:=-300; CLIM.Points[0].Y:=650;
CLIM.Points[1].X:=-50 ; CLIM.Points[1].Y:=650;
CLIM.Points[2].X:= 200; CLIM.Points[2].Y:=200;
CLIM.Points[3].X:= 300; CLIM.Points[3].Y:=200;
CLIM.Points[4].X:= 500; CLIM.Points[4].Y:=200;
CLIM.InitOK:=TRUE;
LogEv(EL_Wrn,EO_CAL,ID,1,'Climatic_default');
END_ACTION

(* POU Plant_Objects/obj_CAL_MGK_2_WOCK, ST *)
FUNCTION_BLOCK obj_CAL_MGK_2_WOCK
(* === CALDAIA VIESSMAN via LON ===
   v1.0[16/04/15] - Versioning
*)
VAR_INPUT
	(* Settings *)
	ID				: BYTE;
	(* Controls *)
	Run				: BOOL;
	RunAcs			: BOOL;


	(* LON Status *)
	ModuleState	  : DWORD;
	(*** LON to CAL ***)




	nvoVorhanden: typSnvtSwitch;
	nvoAlarm:typSnvtCount;
	nvoBoilerMode:typSnvtCount;
	nvoModDegree:typSnvtLevPercent;

	nvoTempBoiler: typSnvtTemp;
	nvoTempHeader: typSnvtTemp;
	nvoTempReturn: typSnvtTemp;
	nvoTempDHW: typSnvtTemp;
	nvoTempOut: typSnvtTemp;

	nvoStateAct:typSnvtState;
	novPressure:typSnvtPress;


	BM_nvoVorhanden: typSnvtSwitch;
	BM_nvoAlarm:typSnvtCount;

	BM_nvoTempRoom: typSnvtTemp;
	BM_nvoSetDHW: typSnvtTemp;
	BM_nvoModeHC:typSnvtCount;
	BM_nvoModeDHW:typSnvtCount;
	BM_nvoTimeHC:typSnvtCount;
	BM_nvoTimeDHW:typSnvtCount;
	BM_nvoSet: typSnvtTemp;
	BM_nvoRed: typSnvtTemp;

	BM_nviSetDHW: typSnvtTemp;
	BM_nviModeHC:typSnvtCount;
	BM_nviModeDHW:typSnvtCount;
	BM_nviTimeHC:typSnvtCount;
	BM_nviTimeDHW:typSnvtCount;
	BM_nviSet: typSnvtTemp;
	BM_nviRed: typSnvtTemp;

	CheckMoreno: typSnvtTemp;


	(* Node inputs *)
	NO_Request    : typSnvtObjRequest;
	NO_TimeSet    : typSnvtTimeStamp;
	NO_AlarmSet   : typSnvtAlarm;
	(* Domestic hot water controller *)
	DHW_ModeSet   : typSnvtHvacMode;
	DHW_SetPoint  : typSnvtTempP;
	(* Central flow demand manager *)
	CFD_SetEnable : typSnvtSwitch;
	CFD_SetMode   : typSnvtHvacMode;
	CFD_SetPoint  : typSnvtTempP;
	(* LON From CAL *)
	NO_Status     : typSnvtObjStatus;
	NO_Alarm      : typSnvtAlarm;
	NO_RlyState   : typSnvtState;
	DHW_ActTemp   : typSnvtTempP;			(* Actual DHW temperature *)
	DHW_SetTemp   : typSnvtTempP;			(* Actual temperature set point *)
	CFD_GetEnable : typSnvtSwitch;
	CFD_Temp      : typSnvtTempP;
	CFD_SetTemp   : typSnvtTempP;

	Temp_S01: INT;
	Temp_S02: INT;
	Temp_S03: INT;
	Temp_S04: INT;



	SetPointManuale: INT; 			(* SetPoint forazato in manuale escludendo la curva di carico *)
	AbilitaSetPointManuale : BOOL ; (* Abilita il funzionamento col set point Manaule Escludendo la curva cliamtica *)
	OffsetBoost: INT;

END_VAR
VAR_IN_OUT
	CLIM		  : typ_Clima;
END_VAR
VAR_OUTPUT
	Curve_Temp	: INT;

	(* Status *)
	Status_Log	: BYTE;
	Status_Vis 	: DWORD;
END_VAR
VAR
	InitOK		: BOOL;
	UpdateOK	: BOOL;
	fAlarm		: BOOL;
	fAlarmBUS	: BOOL;
	fWarning	: BOOL;

	Curve 		: CHARCURVE;
	Curve_Err 	: BYTE;

	Timer1		: TON  := ( PT:=T#5s);		(* Refresh timer for output vars *)

	OLDAllarme: INT;

	TONDelayCheckLON: TON;
	fFaultCheckLON		:	FLT_EVENT;

END_VAR
(* Check initialization *)
(*IF NOT InitOK THEN Init(); END_IF*)

(* le temperature nella caldaia sono in gradi kelvin quindi si deve offsettare tutto a1 - 2740 *)

(* recupero temperature richieste *)

	Temp_S01:=nvoTempOut.wSnvtTemp-2740;
	Temp_S02:=nvoTempBoiler.wSnvtTemp-2740;
	Temp_S03:= nvoTempReturn.wSnvtTemp-2740;
	Temp_S04:=nvoTempDHW.wSnvtTemp-2740;


(* Check LON connection *)
(*
...
*)

(* Check state *)
IF nvoAlarm.wSnvtCount<>OLDAllarme AND ( nvoAlarm.wSnvtCount <132 AND  nvoAlarm.wSnvtCount>1 )THEN
		LogEv(EL_Alarm,EO_CAL,ID,5,CONCAT('Allarme_Caldaia_',INT_TO_STRING( nvoAlarm.wSnvtCount ) ));
		OLDAllarme:=nvoAlarm.wSnvtCount;
		fAlarm:=TRUE;
END_IF

IF nvoAlarm.wSnvtCount= 0 AND fAlarm THEN
		LogEv(EL_LOg,EO_CAL,ID,6,'Allarme_Caldaia_Rientrato');
		OLDAllarme:=nvoAlarm.wSnvtCount;
		fAlarm:= FALSE;
END_IF



(* Check climatic setup *)
IF NOT CLIM.InitOK THEN Clima_Default(); END_IF;
(* Calculate Setpoint *)
Curve(	IN:= T_AMB,	N:= 5, P:= CLIM.Points,
		OUT=> Curve_Temp, ERR=> Curve_Err );
IF Curve_Err>0 THEN
	IF NOT fWarning THEN
		fWarning:=TRUE;
		LogEv(EL_Wrn,EO_CAL,ID,2,'Climatic_Error');
	END_IF
ELSE
	fWarning:=FALSE;
END_IF



(*
(* Scelta del set point della cladaia o vien preso dalla curva cliamtica o da un riferimento esterno *)
IF AbilitaSetPointManuale THEN
	CFD_SetPoint.iSnvtTempP:=(SetPointManuale+OffsetSetPointManuale+OffsetBoost)*10 ;
ELSE
	CFD_SetPoint.iSnvtTempP:=(Curve_Temp+OffsetBoost)*10;
END_IF
*)


(* Attivazione caldaia *)
IF Run   THEN

	BM_nviModeHC.wSnvtCount:=2;		(* 12.4.1 Circuito riscaldamento diretto/miscelato Esercizio automatico  *)

ELSE
	BM_nviModeHC.wSnvtCount:=0;		(* 12.4.1 Circuito riscaldamento diretto/miscelato Standby  *)

END_IF


(* Attivazione caldaia *)
IF THER04.run THEN

	BM_nviModeDHW.wSnvtCount:=2;		(* 12.4.1 Circuito riscaldamento diretto/miscelato Esercizio automatico  *)

ELSE
	BM_nviModeDHW.wSnvtCount:=0;		(* 12.4.1 Circuito riscaldamento diretto/miscelato Standby  *)

END_IF

(* imposo il set point della temperatura dell'acqua calda sanitaria *)
(* fisso in caldaia
CAL01.BM_nviSetDHW.wSnvtTemp:=THER04.SetPoint+2740;
*)




(* Controllo sul comando  Scritto e letto dalla Caldaia  *)

TONDelayCheckLON(IN:=BM_nviModeHC.wSnvtCount<>BM_nvoModeHC.wSnvtCount,PT:=t#3m);
fFaultCheckLON(IN:=TONDelayCheckLON.Q);

IF fFaultCheckLON.EVH THEN
	LogEv(EL_Wrn,EO_CAL,ID,7,'Errore_Comando_Caldaia');
END_IF

IF fFaultCheckLON.EVL THEN
	LogEv(EL_Log,EO_CAL,ID,9,'Comando_Caldaia_Caldaia_OK');
END_IF

fAlarmBUS := TONDelayCheckLON.Q;






(* Status color *)
   IF fAlarm OR fAlarmBUS	THEN Status_Log:=2; Status_Vis:=COLOR_RED;
ELSIF fWarning 		   		THEN Status_Log:=1; Status_Vis:=COLOR_YELLOW;
              				ELSE Status_Log:=0; Status_Vis:=SEL(Run,16#006000,16#20F020);
END_IF
END_FUNCTION_BLOCK
ACTION AddLogData:
Logger.s1:=INSERT('&CAL=',BYTE_TO_STRING(ID),4);
IF ID<10 THEN Logger.s1:=INSERT(Logger.s1,'0',4); END_IF

Logger.s1:=CONCAT(Logger.s1,'0'); (*INT_TO_STRING(CFD_SetPoint.iSnvtTempP/10)); *)
Logger.s1:=CONCAT(Logger.s1,';');
Logger.s1:=CONCAT(Logger.s1,SEL(run,'0','100'));
Logger.s1:=CONCAT(Logger.s1,';');

Logger.s1:=CONCAT(Logger.s1,WORD_TO_STRING(Status_Log));

Logger.s1:=CONCAT(Logger.s1,';');
Logger.s1:=CONCAT(Logger.s1,'0'); (*(OffsetSetPointManuale)); *)
Logger.s1:=CONCAT(Logger.s1,';');
Logger.s1:=CONCAT(Logger.s1,INT_TO_STRING(nvoModDegree.iSnvtLevPercent/204)); (*(CFD_GetEnable.bValue/2)); (* Potenza Caldaia *) *)
Logger.s1:=CONCAT(Logger.s1,';');
Logger.s1:=CONCAT(Logger.s1,SEL(BM_nvoModeHC.wSnvtCount<>0,'0','1'))  ; (*   INT_TO_STRING((BM_nvoModeHC.wSnvtCount)); (*  CFD_GetEnable.siState)); *)	(* Presenza Fiamma *) *)
Logger.s1:=CONCAT(Logger.s1,';');
Logger.s1:=CONCAT(Logger.s1,INT_TO_STRING(Temp_S02)); (*.iSnvtTempP/10)); 	(* Temp. Mandata da Caldaia*) *)
Logger.s1:=CONCAT(Logger.s1,';');
Logger.s1:=CONCAT(Logger.s1,'1');	 									(* Temp. Tipo Caldaia Sempre in questo punto
																				0 = > Albino
																				1 = > Caldaia con Protocollo LON
																				2 = > comandi digitali senza set point *)
Logger.s1:=CONCAT(Logger.s1,';');
Logger.s1:=CONCAT(Logger.s1,'0');	 									(* Manual Mode *)
	


ADDSTRING(ADR(Logger.TData), ADR(Logger.s1), Logger.TLen);
END_ACTION
ACTION Clima_Default:
IF CLIM.Points[0].X=0 THEN
CLIM.Points[0].X:=-300; CLIM.Points[0].Y:=770;
CLIM.Points[1].X:=-70 ; CLIM.Points[1].Y:=770;
CLIM.Points[2].X:= 80;  CLIM.Points[2].Y:=520;
CLIM.Points[3].X:= 200; CLIM.Points[3].Y:=300;
CLIM.Points[4].X:= 500; CLIM.Points[4].Y:=250;
END_IF
CLIM.InitOK:=TRUE;
LogEv(EL_Wrn,EO_CAL,ID,1,'Climatic_default');
END_ACTION
ACTION Heartbeat:
(* Call this at same cycle of LON execution call *)
Timer1(IN:=NOT Timer1.Q,PT:=T#1m);

NO_TimeSet.bDay := SYS.Time_Day;
NO_TimeSet.bMonth := SYS.Time_Month;
NO_TimeSet.iYear := SYS.Time_Year;
NO_TimeSet.bHour := SYS.Time_Hour;
NO_TimeSet.bMinute := SYS.Time_Minute;

NO_TimeSet.bStatusInformation:=SEL(Timer1.Q,0,16#80);
CFD_SetPoint.bStatusInformation:=SEL(Timer1.Q,0,16#80);		(* Re-trigger transmission every 60s *)
CFD_SetMode.bStatusInformation:=SEL(Timer1.Q,0,16#80);
(*CFD_SetEnable.bStatusInformation:=SEL(Timer1.Q,0,16#80);*)
END_ACTION
ACTION Init:
CFD_SetEnable.bValue:=0;

CFD_SetEnable.siState:=BYTE_TO_SINT(16#FF); (* Default value: AUTO *)

CFD_SetMode.bSnvtHvacMode:=16#FF; (* Default value: AUTO *)

(*CAL01.CFD_SetPoint.iSnvtTempP:=0; (* Default temperature: 0°C *)*)

(* End initialization *)
InitOK:=TRUE;
END_ACTION

(* POU Plant_Objects/obj_CIR, ST *)
FUNCTION_BLOCK obj_CIR

(* === CIRCOLATORE STANDARD ===
   v1.0[16/04/15] - Versioning
   v1.1[11/08/15] - Added status reconstruction
*)
VAR CONSTANT
	SampleNr		: BYTE := 120;	(* 1 minute of observation *)
END_VAR
VAR_INPUT
	(* Settings *)
	ID				: BYTE;
	ExtStatus		: BOOL;	(* TRUE: external status signal input available, FALSE: no external status input *)

	(* Physical inputs (Force) *)
	CIR_RUN_REQ		: BOOL; (* External run request (no heat or cold requested) *)
	CIR_STOP_REQ	: BOOL; (* External stop request (has priority over RUN signals!) *)

	(* Physical inputs (Feedback) *)
	Pump_AL			: BOOL; (* Pump Alarm *)
	Pump_ST			: BOOL; (* Pump Status *)
	Pump_AUTO		: BOOL; (* Pump Auto/Manual *)

	(* Controls *)
	OnOff			: BOOL;	(* On/Off from chrono *)
	InitOK			: BOOL;


	(* Input temperature needed if no real feedback about status is available *)
	Tprobe		:	INT;
END_VAR
VAR_OUTPUT
	CIR_EN			: BOOL;

	Ctrl_Run		: BOOL;		(* Logical status of the device: 0: Not running (switched off), 1: running *)
	Run				: BOOL;		(* Real status *)

	Status_Log		: WORD;
	Status_Vis		: DWORD;
END_VAR
VAR
	CIR_AUTO	: 	BOOL; (* Auto/Manual input signal *)
	Pump_En		:	BOOL;

	(* Filters *)
	fPump_ST	: 	FLT_TAP := (INITEV:=FALSE);
	fPump_En	:	FLT_EVENT;
	fCIR_AUTO	:	FLT_TAP;
	fStatus		:	FLT_EVENT;
	fStatusFault:	BOOL;

	(* Timer manage switch on/off delay *)
	Delay		: 	TONOF;

	(* Alarm and Warning counters *)
	AlarmCtr	:	BYTE;
	WarningCtr	:	BYTE;

	(* Filers on alarms and faults *)
	AlarmHw		:	FLT_TAP := (INITEV:=FALSE);

	(* Variables for status reconstruction *)
	aTprobe		:	ARRAY [1..SampleNr] OF INT;
	sample		:	BYTE;
	Tmean		:	INT;
	sum			:	INT;
	i			:	BYTE;
END_VAR



VAR_INPUT RETAIN
		(* Timings *)
	OnDelay		:	TIME;	(* Switch on delay *)
	OffDelay	:	TIME;	(* Switch off delay *)

END_VAR
Init();


StatusRebuild();
(* Check alarms and warnings *)
CheckFault();

PumpManager();

IF AlarmCtr>0 THEN
	Status_Log := 2;
	Status_Vis := COLOR_RED;
ELSIF WarningCtr>0 OR fPump_ST.OUT THEN
	Status_Log := 1;
	Status_Vis := COLOR_YELLOW;
ELSE
	Status_Log := 0;
	Status_Vis := COLOR_GREEN;
END_IF
END_FUNCTION_BLOCK
ACTION AddLogData:
Logger.s1:=INSERT('&CIR=',BYTE_TO_STRING(ID),4);
IF ID<10 THEN Logger.s1:=INSERT(Logger.s1,'0',4); END_IF

Logger.s1:=CONCAT(Logger.s1,SEL(Pump_En,'0','100'));		Logger.s1:=CONCAT(Logger.s1,';');

Logger.s1:=CONCAT(Logger.s1,WORD_TO_STRING(Status_Log));
Logger.s1:=CONCAT(Logger.s1,';');
Logger.s1:=CONCAT(Logger.s1,SEL(CIR_RUN_REQ,'0','100'));
Logger.s1:=CONCAT(Logger.s1,';');
Logger.s1:=CONCAT(Logger.s1,SEL(CIR_STOP_REQ,'0','100'));



ADDSTRING(ADR(Logger.TData), ADR(Logger.s1), Logger.TLen);
END_ACTION
ACTION CheckFault:
(*** ALARMS ***)

(* Hardware alarm (physical input *)
AlarmHw(IN:=Pump_AL);

IF AlarmHw.EVH THEN
	LogEv(EL_Alarm,EO_CIR,ID,3,'');
	AlarmCtr := AlarmCtr + 1;
END_IF

IF AlarmHw.EVL THEN
	LogEv(EL_Log,EO_CIR,ID,4,'');
	AlarmCtr := SEL(AlarmCtr=0, AlarmCtr-1, 0);
END_IF

IF ExtStatus THEN
	fPump_ST(IN:=(Pump_ST<>CIR_EN));

	IF fPump_ST.EVH THEN
		IF Pump_AUTO THEN
			LogEv(SEL(Pump_ST,EL_Alarm,EL_Wrn),EO_CIR,ID,SEL(Pump_ST,5,6),'');
		ELSE
			LogEv(EL_Wrn,EO_CIR,ID,SEL(Pump_ST,1,2),'');
		END_IF
	END_IF

ELSE
	fPump_ST(IN:=fStatusFault);

	IF fPump_ST.EVH THEN
		IF Pump_AUTO THEN
			LogEv(SEL(OnOff,EL_Alarm,EL_Wrn),EO_CIR,ID,SEL(OnOff,5,6),'');
		ELSE
			LogEv(EL_Wrn,EO_CIR,ID,SEL(OnOff,1,2),'');
		END_IF
	END_IF
END_IF
END_ACTION
ACTION Init:
IF NOT InitOK THEN

	Pump_En := FALSE;

	InitOK := TRUE;

END_IF
END_ACTION
ACTION PumpManager:
(* Aggiornamento in tempo reale dei TON e TOFF funzionamento Pompa *)

Delay.PT_OF := OffDelay;
Delay.PT_ON := OnDelay + WORD_TO_TIME(1000*ID);




(* Verify if in Auto or Manual mode *)
fCIR_AUTO(IN:=Pump_AUTO);

IF fCIR_AUTO.EVH THEN
	LogEv(EL_Log,EO_CIR,ID,8,'CIR_Auto');
	WarningCtr := SEL(WarningCtr=0, WarningCtr-1,0);
END_IF

(* Manual -> Keep switched on *)
IF fCIR_AUTO.EVL THEN
	LogEv(EL_Wrn,EO_CIR,ID,7,'CIR_Manual');
	WarningCtr := WarningCtr + 1;

	(* Switch on pump *)
	Pump_En := TRUE;
END_IF

(* Verify if OnOff is changed *)
Ctrl_Run := OnOff;

(* Check switch on or switch off delay *)
Delay(IN:=Ctrl_Run);

(* Do these instructions only if in AUTO mode *)
IF Pump_AUTO THEN
	(* If priority request *)
	IF CIR_STOP_REQ THEN Pump_En := FALSE;
	ELSIF CIR_RUN_REQ THEN Pump_En := TRUE;
	ELSE Pump_En := Delay.OUT;
	END_IF

	(* Set RUN signal (for external objects) *)
	IF AlarmHw.OUT THEN
		Run:=FALSE;
	ELSE
		Run:=Pump_En;
	END_IF
END_IF

(* Set value on physical outuput! *)
CIR_EN := Pump_En;
END_ACTION
ACTION StatusRebuild:
IF NOT ExtStatus THEN
	(* Check every 20 seconds *)
	IF  sample<sampleNr THEN
	
		aTprobe[sample] := Tprobe;
		sample := sample + 1;
	
	ELSE
	
		SHIFT_ARRAY(ADR(aTprobe),SampleNr);
	
		FOR i:=1 TO SampleNr BY 1 DO
			sum := sum + aTprobe[i];
		END_FOR
	
		Tmean := sum/SampleNr;
	
		(* CIR should be on but revealed temperature is decreasing *)
		IF OnOff AND (Tprobe<aTprobe[1]) THEN
			fStatusFault := TRUE;
		ELSE
			fStatusFault := FALSE;
		END_IF
	
		(* CIR should be off but revealed temperature is increasing *)
		IF NOT OnOff AND (Tprobe>aTprobe[1]) THEN
			fStatusFault := TRUE;
		ELSE
			fStatusFault := FALSE;
		END_IF
	END_IF
END_IF
END_ACTION

(* POU Utils Functions/TONOF, ST *)
FUNCTION_BLOCK TONOF
VAR_INPUT
	IN		: BOOL;
	PT_ON	: TIME; (* time to pass, before OUT is set *)
	PT_OF	: TIME; (* time to pass, before OUT is reset *)
END_VAR
VAR_OUTPUT
	OUT		: BOOL;
END_VAR
VAR
	timer	: TON;
END_VAR
IF IN<>OUT THEN
	timer(IN:=TRUE,PT:=SEL(IN,PT_OF,PT_ON));
	IF timer.Q THEN OUT:=IN; END_IF
ELSE
	timer(IN:=FALSE);
END_IF
END_FUNCTION_BLOCK

(* POU Plant_Objects/obj_CRON_EDITOR_01, ST *)
FUNCTION_BLOCK obj_CRON_EDITOR_01
(* === EDITOR CRONOGRAFO ===
   v1.0[16/04/15] - Versioning
   v1.1[19/05/15] - Create empty profile when not found
*)
VAR_INPUT

	(* Common selections *)
	CN_Sel:			BYTE:=1;
	CN_Act:			BYTE;
	CN_YSel:		WORD:=2015;
	CN_YAct:		WORD;

	(* Profile editor *)
	PR_Sel: 		BYTE:=1;
	PR_Act:			BYTE;
	PR_TT:			REAL;
	PR:				typ_Cron_Profile;
	(* Profile signals *)
	PR_Load:		BOOL;
	PR_Save:		BOOL;

	(* Calendar editor *)
	CA_Sel:			BYTE:=1; (* Calendar month selected *)
	CA_Act:			BYTE;    (* Calendar month active *)
	CA_DayF:		BYTE:=0;
	CA_DayL:		BYTE:=31;
	CA_TPR:			BYTE;
	CA:				typ_Cron_Calendar; (* Only used for first 32 entries *)
	(* Calendar signals *)
	CA_Load:		BOOL;
	CA_Save:		BOOL;

	(* Jolly editor *)
	JL:				ARRAY[0..9] OF typ_Cron_Jolly;
	(* Jolly signals *)
	JL_Load:		BOOL;
	JL_Save:		BOOL;

END_VAR
VAR_OUTPUT
	Message		: STRING;
END_VAR
VAR
	sFileName	: STRING;
	sFileMode	: STRING;
	hFile		: DWORD;
	Buf			: ARRAY[0..512] OF BYTE; (* AVOID THIS!! *)

	i			: WORD;
	ver			: BYTE;
	r1			: BOOL;
	r2			: DWORD;

	x: INT;
	maxProfili: INT;

	sFileNameOld	: STRING;
	sFileModeOld		: STRING;
	hFileOld			: DWORD;




	strAppoggio: STRING;
	FileGiaCreato: BOOL;
	fileCopiato: UDINT;

	tempMultiAnnoMax:INT;
	tempMultiAnnoIndex:INT;
	TEMP_MULTIANNO_MAX_DELTA:INT:=5;
	tempRicercaFileAnno:INT;
	tempAnno:INT;
	tempTrovato:BOOL;
END_VAR
IF PR_Load THEN PR_Load_Exe();
	PR_Load:=FALSE;
END_IF
IF PR_Save THEN
PR_Save_Exe();
PR_Save:=FALSE;
END_IF
IF CA_Load THEN
CA_Load_Exe();
CA_Load:=FALSE;
END_IF
IF CA_Save THEN
CA_Save_Exe();
CA_Save:=FALSE;
END_IF
IF JL_Load THEN
JL_Load_Exe();
JL_Load:=FALSE;
END_IF
IF JL_Save THEN
 JL_Save_Exe();
 JL_Save:=FALSE;
 END_IF
END_FUNCTION_BLOCK
ACTION CA_Load_Exe:
sFileMode:='r';
FileOpen();

IF hFile<>0 THEN

	(* Read calendar month *)
	FOR i := 0 TO 31 DO
		r1:=SysFileSetPos(File:=hFile, Pos:=(1024 + ((CA_Sel-1)*32 + i)*4));
		r2:=SysFileRead(File:=hFile, Buffer:=ADR(CA.Profile[i]), Size:=1);
	END_FOR

	(* Close file *)
	SysFileClose(File:=hFile);

	(* Validate data *)
	CA_Act :=CA_Sel;
	CN_Act :=CN_Sel;
	CN_YAct:=CN_YSel;

	Message:='Calendar load OK';

END_IF
END_ACTION
ACTION CA_Save_Exe:
sFileMode:='a';
FileOpen();

IF hFile<>0 THEN

	(* Write calendar month *)
	FOR i := 0 TO 31 DO
		r1:=SysFileSetPos(File:=hFile, Pos:=(1024 + ((CA_Sel-1)*32 + i)*4));
		r2:=SysFileGetPos(hFile);
		r2:=SysFileWrite(File:=hFile, Buffer:=ADR(CA.Profile[i]), Size:=1);
	END_FOR

	(* Close file *)
	SysFileClose(File:=hFile);

	Message:='Calendar save OK';

	(* db commentato! non salva i profili, ma solo il profilo corrente, che può anche essere modificato!*)
          (*PR_Save_exe();*)
	(* nel salvare il calendario aggiorno anche i profili così ho il file completo dei profili *)


END_IF

IF hFile<>0 THEN SysFileClose(File:=hFile); END_IF (*diego add*)
END_ACTION
ACTION FileOpen:
(* Create current filename 'yyyyCRnn.DAT' *) (* creo il nome del file da aparire *)
sFileName:=CONCAT(FilesPath,WORD_TO_STRING(CN_YSel));
sFileName:=CONCAT(STR1:=sFileName, STR2:='CR');
IF CN_Sel<10 THEN
sFileName:=CONCAT(STR1:=sFileName, STR2:='0');
END_IF
sFileName:=CONCAT(STR1:=sFileName, STR2:=BYTE_TO_STRING(CN_Sel));
sFileName:=CONCAT(STR1:=sFileName, STR2:='.DAT');


(* Apro il fiel in lettura per verificare se è presente altrimenti devo crearne uno nuovo a duplicare quello dell'anno precedente - apro 1  *)
hFile:=SysFileOpen(FileName:=sFileName, Mode:='r');
FileGiaCreato:=FALSE;

tempAnno:=CN_YSel;
tempTrovato:=FALSE;

(* File non trovato da creare  *)
IF hFile=0 THEN

	 (*cerco i file precendti: dall'anno prima fino a - TEMP_MULTIANNO_MAX_DELTA*)
	 tempRicercaFileAnno:=1;

	WHILE tempRicercaFileAnno<=TEMP_MULTIANNO_MAX_DELTA AND NOT tempTrovato DO


		strAppoggio:=INT_TO_STRING(tempAnno);
		(* Verifico se esite un file da cui partire *)
		StrAppoggio:=WORD_TO_STRING(STRING_TO_WORD(strAppoggio)-tempRicercaFileAnno);
		sFileNameOld:=CONCAT(FilesPath,StrAppoggio);

		sFileNameOld:=CONCAT(STR1:=sFileNameOld, STR2:='CR');
		IF CN_Sel<10 THEN
			sFileNameOld:=CONCAT(STR1:=sFileNameOld, STR2:='0');
		END_IF
		sFileNameOld:=CONCAT(STR1:=sFileNameOld, STR2:=BYTE_TO_STRING(CN_Sel));
		sFileNameOld:=CONCAT(STR1:=sFileNameOld, STR2:='.DAT');

		(* Apro il file in lettura per la verifica della presenza del file da copiare  *)
		hFileold:=SysFileOpen(FileName:=sFileNameOld, Mode:='r');

		IF hFileold<>0 THEN

			tempTrovato:=TRUE;

			fileCopiato:=SysFileCopy(sFileName,sFileNameold);

    		   	FileGiaCreato:=fileCopiato<>0;

			IF FileGiaCreato THEN
				Message:='File Sorgente/copia  trovato - file Copiato';
			ELSE
				Message:='File Sorgente/copia  trovato - file NON Copiato';
			END_IF


			(* Chiudo il file aperto per la verifica del file presente *)
			SysFileClose(File:=hFile);
			(* Chiudo il file aperto in lettura per la verifica della presenza del file da copiare  *)
			SysFileClose(File:=hFileold);

		END_IF

		tempRicercaFileAnno:=tempRicercaFileAnno+1;

	END_WHILE

	(* se non ho trovato nessun file..lo creo vuoto*)
	IF tempTrovato=FALSE THEN   (* file non trovato quindi devo crearne uno nuovo *)

			(* Create empty file *)
			hFile:=SysFileOpen(FileName:=sFileName, Mode:='w');
			MEMCLR(pDestinationAddress:=ADR(Buf), BytesToClear:=SIZEOF(Buf));
			FOR i := 0 TO 10239 BY 512 DO
				SysFileWrite(File:=hFile, Buffer:=ADR(Buf), Size:=512);
			END_FOR

			Buf[0]:=1;
			SysFileSetPos(File:=hFile, Pos:=0);
			SysFileWrite(File:=hFile, Buffer:=ADR(Buf), Size:=1);

			(* Chiudo il file aperto per la verifica del file presente *)
			SysFileClose(File:=hFile);
			(* Chiudo il file aperto in lettura per la verifica della presenza del file da copiare  *)
			SysFileClose(File:=hFileold);

			Message:='File Sorgente/copia non trovato-file Vuoto';

	END_IF


ELSE

	(* Chiudo il file aperto per la verifica del file presente *)
	SysFileClose(File:=hFile);

END_IF




(* Apro il file per permettere la scrittura o la lettura del file da parte delle altre action . la chiusura del file è delegata alle Action *)
hFile:=SysFileOpen(FileName:=sFileName, Mode:=sFileMode);
END_ACTION
ACTION JL_Load_Exe:
sFileMode:='r';
FileOpen();

IF hFile<>0 THEN

	(* Read jolly *)
	r1:=SysFileSetPos(File:=hFile, Pos:=512);
	r2:=SysFileRead(File:=hFile, Buffer:=ADR(JL), Size:=SIZEOF(JL));

	(* Close file *)
	SysFileClose(File:=hFile);

	(* Validate data *)
	CN_Act:=CN_Sel;
	CN_YAct:=CN_YSel;

	Message:='Jolly load OK';

END_IF
END_ACTION
ACTION JL_Save_Exe:
sFileMode:='a';
FileOpen();

IF hFile<>0 THEN

	(* Write selected profile *)
	r1:=SysFileSetPos(File:=hFile, Pos:=512);
	r2:=SysFileWrite(File:=hFile, Buffer:=ADR(JL), Size:=SIZEOF(JL));

	(* Close file *)
	SysFileClose(File:=hFile);

	Message:='Jolly save OK';

END_IF
END_ACTION
ACTION PR_Load_Exe:
sFileMode:='r';
FileOpen();

IF hFile<>0 THEN

	(* Read selected profile *)
	r1:=SysFileSetPos(File:=hFile, Pos:=(3072 + 512*PR_Sel));
	r2:=SysFileRead(File:=hFile, Buffer:=ADR(PR), Size:=SIZEOF(PR));

	(* Close file *)
	SysFileClose(File:=hFile);

	(* Validate data *)
	PR_Act:=PR_Sel;
	CN_Act:=CN_Sel;
	CN_YAct:=CN_YSel;

	Message:='Profile load OK';

END_IF
END_ACTION
ACTION PR_Save_Exe:
sFileMode:='a';
FileOpen();

IF hFile<>0 THEN

		(* Write selected profile *)
		r1:=SysFileSetPos(File:=hFile, Pos:=(3072 + 512*PR_Sel));
		r2:=SysFileWrite(File:=hFile, Buffer:=ADR(PR), Size:=SIZEOF(PR));

		(* Close file *)
		SysFileClose(File:=hFile);

		Message:='Profile save OK';

END_IF

IF hFile<>0 THEN SysFileClose(File:=hFile); END_IF (*diego add*)
END_ACTION
ACTION PR_Save_Exe_Multi:
(*eseguo  salvataggio profilo per l'anno corrente del CronoEditor - quello indicato da CN_YSel*)
CronEd.PR_Save_Exe();

